LIN {X 0,Y 298.713,Z 404.512,A -85,B 0,C 180,E1 -16393.955,E2 -16393.955} C_VEL
LIN {X 0,Y 299.708,Z 394.679,A -85,B 0,C 180,E1 -16396.344,E2 -16396.344} C_VEL
LIN {X 0,Y 300.926,Z 384.674,A -85,B 0,C 180,E1 -16398.379,E2 -16398.379} C_VEL
LIN {X 0,Y 302.379,Z 372.804,A -85,B 0,C 180,E1 -16400.404,E2 -16400.404} C_VEL
LIN {X 0,Y 303.908,Z 359.25,A -85,B 0,C 180,E1 -16402.329,E2 -16402.329} C_VEL
LIN {X 0,Y 305.452,Z 345.622,A -85,B 0,C 180,E1 -16403.925,E2 -16403.925} C_VEL
LIN {X 0,Y 306.858,Z 331.853,A -85,B 0,C 180,E1 -16405.251,E2 -16405.251} C_VEL
LIN {X 0,Y 308.322,Z 315.885,A -85,B 0,C 180,E1 -16406.482,E2 -16406.482} C_VEL
LIN {X 0,Y 309.428,Z 299.28,A -85,B 0,C 180,E1 -16407.46,E2 -16407.46} C_VEL
LIN {X 0,Y 310.381,Z 282.456,A -85,B 0,C 180,E1 -16408.156,E2 -16408.156} C_VEL
LIN {X 0,Y 315.944,Z 175.453,A -85,B 0,C 180,E1 -16411.633,E2 -16411.633} C_VEL
LIN {X 0,Y 298.499,Z 134.359,A -85,B 0,C 180,E1 -16414.507,E2 -16414.507} C_VEL
LIN {X 0,Y 298.417,Z 133.938,A -85,B 0,C 180,E1 -16414.556,E2 -16414.556} C_VEL
LIN {X 0,Y 298.4,Z 133.941,A -85,B 0,C 180,E1 -16417.761,E2 -16417.761} C_VEL
LIN {X 0,Y 298.349,Z 133.947,A -85,B 0,C 180,E1 -16421.268,E2 -16421.268} C_VEL
LIN {X 0,Y 298.356,Z 133.922,A -85,B 0,C 180,E1 -16425.035,E2 -16425.035} C_VEL
LIN {X 0,Y 298.35,Z 133.935,A -85,B 0,C 180,E1 -16428.921,E2 -16428.921} C_VEL
LIN {X 0,Y 298.4,Z 133.933,A -85,B 0,C 180,E1 -16432.24,E2 -16432.24} C_VEL
LIN {X 0,Y 298.41,Z 133.92,A -85,B 0,C 180,E1 -16435.581,E2 -16435.581} C_VEL
LIN {X 0,Y 298.379,Z 133.936,A -85,B 0,C 180,E1 -16438.789,E2 -16438.789} C_VEL
LIN {X 0,Y 298.413,Z 133.928,A -85,B 0,C 180,E1 -16441.899,E2 -16441.899} C_VEL
LIN {X 0,Y 298.417,Z 133.926,A -85,B 0,C 180,E1 -16444.918,E2 -16444.918} C_VEL
LIN {X 0,Y 298.395,Z 133.941,A -85,B 0,C 180,E1 -16447.862,E2 -16447.862} C_VEL
LIN {X 0,Y 298.463,Z 133.922,A -85,B 0,C 180,E1 -16450.752,E2 -16450.752} C_VEL
LIN {X 0,Y 298.514,Z 133.924,A -85,B 0,C 180,E1 -16454.991,E2 -16454.991} C_VEL
LIN {X 0,Y 298.526,Z 133.999,A -85,B 0,C 180,E1 -16456.297,E2 -16456.297} C_VEL
LIN {X 0,Y 302.475,Z 145.498,A -85,B 0,C 180,E1 -16459.094,E2 -16459.094} C_VEL
LIN {X 0,Y 310.955,Z 161.787,A -85,B 0,C 180,E1 -16460.635,E2 -16460.635} C_VEL
LIN {X 0,Y 320.63,Z 183.073,A -85,B 0,C 180,E1 -16462.347,E2 -16462.347} C_VEL
LIN {X 0,Y 323.385,Z 190.184,A -85,B 0,C 180,E1 -16462.842,E2 -16462.842} C_VEL
LIN {X 0,Y 318.857,Z 312.214,A -85,B 0,C 180,E1 -16465.615,E2 -16465.615} C_VEL
LIN {X 0,Y 317.724,Z 327.891,A -85,B 0,C 180,E1 -16466.195,E2 -16466.195} C_VEL
LIN {X 0,Y 316.387,Z 342.225,A -85,B 0,C 180,E1 -16466.971,E2 -16466.971} C_VEL
LIN {X 0,Y 314.797,Z 355.633,A -85,B 0,C 180,E1 -16467.921,E2 -16467.921} C_VEL
LIN {X 0,Y 312.756,Z 369.748,A -85,B 0,C 180,E1 -16469.195,E2 -16469.195} C_VEL
LIN {X 0,Y 310.496,Z 382.746,A -85,B 0,C 180,E1 -16470.648,E2 -16470.648} C_VEL
LIN {X 0,Y 308.101,Z 395.661,A -85,B 0,C 180,E1 -16472.435,E2 -16472.435} C_VEL
LIN {X 0,Y 305.908,Z 406.678,A -85,B 0,C 180,E1 -16474.282,E2 -16474.282} C_VEL
LIN {X 0,Y 303.719,Z 417.119,A -85,B 0,C 180,E1 -16476.392,E2 -16476.392} C_VEL
LIN {X 0,Y 301.643,Z 426.588,A -85,B 0,C 180,E1 -16478.711,E2 -16478.711} C_VEL
LIN {X 0,Y 300.015,Z 434.716,A -85,B 0,C 180,E1 -16481.143,E2 -16481.143} C_VEL
LIN {X 0,Y 298.703,Z 441.439,A -85,B 0,C 180,E1 -16483.608,E2 -16483.608} C_VEL
LIN {X 0,Y 297.604,Z 447.559,A -85,B 0,C 180,E1 -16486.462,E2 -16486.462} C_VEL
LIN {X 0,Y 297.001,Z 451.472,A -85,B 0,C 180,E1 -16488.82,E2 -16488.82} C_VEL
LIN {X 0,Y 296.584,Z 453.996,A -85,B 0,C 180,E1 -16490.821,E2 -16490.821} C_VEL
LIN {X 0,Y 296.399,Z 455.502,A -85,B 0,C 180,E1 -16492.37,E2 -16492.37} C_VEL
LIN {X 0,Y 296.198,Z 457.301,A -85,B 0,C 180,E1 -16495.283,E2 -16495.283} C_VEL
LIN {X 0,Y 296.215,Z 457.762,A -85,B 0,C 180,E1 -16498.328,E2 -16498.328} C_VEL
LIN {X 0,Y 296.405,Z 456.777,A -85,B 0,C 180,E1 -16501.395,E2 -16501.395} C_VEL
LIN {X 0,Y 296.835,Z 454.759,A -85,B 0,C 180,E1 -16504.036,E2 -16504.036} C_VEL
LIN {X 0,Y 297.466,Z 451.962,A -85,B 0,C 180,E1 -16506.435,E2 -16506.435} C_VEL
LIN {X 0,Y 297.135,Z 450.458,A -85,B 0,C 180,E1 -16507.534,E2 -16507.534} C_VEL
LIN {X 0,Y 294.916,Z 447.714,A -85,B 0,C 180,E1 -16509.328,E2 -16509.328} C_VEL
LIN {X 0,Y 293.14,Z 445.205,A -85,B 0,C 180,E1 -16510.759,E2 -16510.759} C_VEL
LIN {X 0,Y 292.687,Z 443.03,A -85,B 0,C 180,E1 -16511.834,E2 -16511.834} C_VEL
LIN {X 0,Y 292.82,Z 442.243,A -85,B 0,C 180,E1 -16512.189,E2 -16512.189} C_VEL
LIN {X 0,Y 294.596,Z 435.357,A -85,B 0,C 180,E1 -16514.833,E2 -16514.833} C_VEL
LIN {X 0,Y 296.759,Z 427.599,A -85,B 0,C 180,E1 -16517.236,E2 -16517.236} C_VEL
LIN {X 0,Y 298.988,Z 419.592,A -85,B 0,C 180,E1 -16519.294,E2 -16519.294} C_VEL
LIN {X 0,Y 301.649,Z 409.459,A -85,B 0,C 180,E1 -16521.469,E2 -16521.469} C_VEL
LIN {X 0,Y 304.318,Z 398.99,A -85,B 0,C 180,E1 -16523.325,E2 -16523.325} C_VEL
LIN {X 0,Y 307.208,Z 386.777,A -85,B 0,C 180,E1 -16525.115,E2 -16525.115} C_VEL
LIN {X 0,Y 310.013,Z 373.338,A -85,B 0,C 180,E1 -16526.716,E2 -16526.716} C_VEL
LIN {X 0,Y 312.66,Z 358.816,A -85,B 0,C 180,E1 -16528.088,E2 -16528.088} C_VEL
LIN {X 0,Y 314.776,Z 345.041,A -85,B 0,C 180,E1 -16529.101,E2 -16529.101} C_VEL
LIN {X 0,Y 316.458,Z 330.282,A -85,B 0,C 180,E1 -16529.935,E2 -16529.935} C_VEL
LIN {X 0,Y 317.811,Z 314.936,A -85,B 0,C 180,E1 -16530.525,E2 -16530.525} C_VEL
LIN {X 0,Y 318.317,Z 302.146,A -85,B 0,C 180,E1 -16530.882,E2 -16530.882} C_VEL
LIN {X 0,Y 315.448,Z 304.886,A -85,B 0,C 180,E1 -16531.197,E2 -16531.197} C_VEL
LIN {X 0,Y 312.655,Z 306.053,A -85,B 0,C 180,E1 -16531.558,E2 -16531.558} C_VEL
LIN {X 0,Y 311.943,Z 306.129,A -85,B 0,C 180,E1 -16531.659,E2 -16531.659} C_VEL
LIN {X 0,Y 308.747,Z 312.307,A -85,B 0,C 180,E1 -16531.919,E2 -16531.919} C_VEL
LIN {X 0,Y 306.255,Z 315.221,A -85,B 0,C 180,E1 -16532.169,E2 -16532.169} C_VEL
LIN {X 0,Y 304.049,Z 316.166,A -85,B 0,C 180,E1 -16532.464,E2 -16532.464} C_VEL
LIN {X 0,Y 302.853,Z 315.629,A -85,B 0,C 180,E1 -16532.674,E2 -16532.674} C_VEL
LIN {X 0,Y 301.938,Z 313.525,A -85,B 0,C 180,E1 -16532.913,E2 -16532.913} C_VEL
LIN {X 0,Y 301.81,Z 312.672,A -85,B 0,C 180,E1 -16532.994,E2 -16532.994} C_VEL
LIN {X 0,Y 300.389,Z 328.503,A -85,B 0,C 180,E1 -16534.166,E2 -16534.166} C_VEL
LIN {X 0,Y 298.938,Z 342.979,A -85,B 0,C 180,E1 -16535.52,E2 -16535.52} C_VEL
LIN {X 0,Y 297.42,Z 356.501,A -85,B 0,C 180,E1 -16537.065,E2 -16537.065} C_VEL
LIN {X 0,Y 295.874,Z 370.051,A -85,B 0,C 180,E1 -16538.944,E2 -16538.944} C_VEL
LIN {X 0,Y 294.385,Z 381.5,A -85,B 0,C 180,E1 -16540.836,E2 -16540.836} C_VEL
LIN {X 0,Y 293.12,Z 392.122,A -85,B 0,C 180,E1 -16542.919,E2 -16542.919} C_VEL
LIN {X 0,Y 291.957,Z 402.502,A -85,B 0,C 180,E1 -16545.359,E2 -16545.359} C_VEL
LIN {X 0,Y 291.111,Z 410.013,A -85,B 0,C 180,E1 -16547.45,E2 -16547.45} C_VEL
LIN {X 0,Y 290.371,Z 418.242,A -85,B 0,C 180,E1 -16550.245,E2 -16550.245} C_VEL
LIN {X 0,Y 289.956,Z 424.764,A -85,B 0,C 180,E1 -16553.039,E2 -16553.039} C_VEL
LIN {X 0,Y 289.765,Z 429.759,A -85,B 0,C 180,E1 -16555.827,E2 -16555.827} C_VEL
LIN {X 0,Y 289.641,Z 433.363,A -85,B 0,C 180,E1 -16558.609,E2 -16558.609} C_VEL
LIN {X 0,Y 289.791,Z 435.684,A -85,B 0,C 180,E1 -16561.389,E2 -16561.389} C_VEL
LIN {X 0,Y 290.122,Z 436.747,A -85,B 0,C 180,E1 -16564.167,E2 -16564.167} C_VEL
LIN {X 0,Y 290.689,Z 436.577,A -85,B 0,C 180,E1 -16566.943,E2 -16566.943} C_VEL
LIN {X 0,Y 291.75,Z 435.204,A -85,B 0,C 180,E1 -16569.707,E2 -16569.707} C_VEL
LIN {X 0,Y 293.145,Z 432.65,A -85,B 0,C 180,E1 -16572.46,E2 -16572.46} C_VEL
LIN {X 0,Y 294.431,Z 429.964,A -85,B 0,C 180,E1 -16574.515,E2 -16574.515} C_VEL
LIN {X 0,Y 296.723,Z 425.209,A -85,B 0,C 180,E1 -16577.221,E2 -16577.221} C_VEL
LIN {X 0,Y 299.687,Z 419.075,A -85,B 0,C 180,E1 -16579.879,E2 -16579.879} C_VEL
LIN {X 0,Y 303.206,Z 411.451,A -85,B 0,C 180,E1 -16582.485,E2 -16582.485} C_VEL
LIN {X 0,Y 306.675,Z 403.431,A -85,B 0,C 180,E1 -16584.723,E2 -16584.723} C_VEL
LIN {X 0,Y 310.706,Z 393.918,A -85,B 0,C 180,E1 -16586.897,E2 -16586.897} C_VEL
LIN {X 0,Y 315.196,Z 382.723,A -85,B 0,C 180,E1 -16589.003,E2 -16589.003} C_VEL
LIN {X 0,Y 319.857,Z 370.152,A -85,B 0,C 180,E1 -16590.959,E2 -16590.959} C_VEL
LIN {X 0,Y 324.749,Z 355.792,A -85,B 0,C 180,E1 -16592.754,E2 -16592.754} C_VEL
LIN {X 0,Y 328.897,Z 342.374,A -85,B 0,C 180,E1 -16594.119,E2 -16594.119} C_VEL
LIN {X 0,Y 332.878,Z 327.973,A -85,B 0,C 180,E1 -16595.307,E2 -16595.307} C_VEL
LIN {X 0,Y 336.634,Z 312.349,A -85,B 0,C 180,E1 -16596.327,E2 -16596.327} C_VEL
LIN {X 0,Y 339.839,Z 296.318,A -85,B 0,C 180,E1 -16597.128,E2 -16597.128} C_VEL
LIN {X 0,Y 354.117,Z 224.063,A -85,B 0,C 180,E1 -16599.946,E2 -16599.946} C_VEL
LIN {X 0,Y 355.571,Z 217.184,A -85,B 0,C 180,E1 -16600.229,E2 -16600.229} C_VEL
LIN {X 0,Y 354.234,Z 214.83,A -85,B 0,C 180,E1 -16602.1,E2 -16602.1} C_VEL
LIN {X 0,Y 353.367,Z 214.935,A -85,B 0,C 180,E1 -16604.275,E2 -16604.275} C_VEL
LIN {X 0,Y 353.324,Z 216.461,A -85,B 0,C 180,E1 -16605.878,E2 -16605.878} C_VEL
LIN {X 0,Y 353.663,Z 218.476,A -85,B 0,C 180,E1 -16607.134,E2 -16607.134} C_VEL
LIN {X 0,Y 354.272,Z 222.512,A -85,B 0,C 180,E1 -16608.612,E2 -16608.612} C_VEL
LIN {X 0,Y 354.554,Z 224.671,A -85,B 0,C 180,E1 -16609.192,E2 -16609.192} C_VEL
LIN {X 0,Y 340.864,Z 295.02,A -85,B 0,C 180,E1 -16611.907,E2 -16611.907} C_VEL
LIN {X 0,Y 335.929,Z 321.398,A -85,B 0,C 180,E1 -16613,E2 -16613} C_VEL
LIN {X 0,Y 331.767,Z 338.526,A -85,B 0,C 180,E1 -16613.902,E2 -16613.902} C_VEL
LIN {X 0,Y 326.822,Z 355.759,A -85,B 0,C 180,E1 -16615.072,E2 -16615.072} C_VEL
LIN {X 0,Y 321.962,Z 371.081,A -85,B 0,C 180,E1 -16616.41,E2 -16616.41} C_VEL
LIN {X 0,Y 316.965,Z 385.854,A -85,B 0,C 180,E1 -16618.037,E2 -16618.037} C_VEL
LIN {X 0,Y 312.28,Z 398.757,A -85,B 0,C 180,E1 -16619.764,E2 -16619.764} C_VEL
LIN {X 0,Y 307.82,Z 410.76,A -85,B 0,C 180,E1 -16621.722,E2 -16621.722} C_VEL
LIN {X 0,Y 303.56,Z 421.893,A -85,B 0,C 180,E1 -16623.903,E2 -16623.903} C_VEL
LIN {X 0,Y 299.527,Z 432.689,A -85,B 0,C 180,E1 -16626.492,E2 -16626.492} C_VEL
LIN {X 0,Y 296.239,Z 441.705,A -85,B 0,C 180,E1 -16629.154,E2 -16629.154} C_VEL
LIN {X 0,Y 293.617,Z 449.164,A -85,B 0,C 180,E1 -16631.87,E2 -16631.87} C_VEL
LIN {X 0,Y 291.114,Z 459.129,A -85,B 0,C 180,E1 -16636.03,E2 -16636.03} C_VEL
LIN {X 0,Y 290.103,Z 464.483,A -85,B 0,C 180,E1 -16638.825,E2 -16638.825} C_VEL
LIN {X 0,Y 289.628,Z 468.472,A -85,B 0,C 180,E1 -16641.628,E2 -16641.628} C_VEL
LIN {X 0,Y 289.433,Z 471.324,A -85,B 0,C 180,E1 -16644.595,E2 -16644.595} C_VEL
LIN {X 0,Y 289.455,Z 472.691,A -85,B 0,C 180,E1 -16647.217,E2 -16647.217} C_VEL
LIN {X 0,Y 289.439,Z 473.009,A -85,B 0,C 180,E1 -16650,E2 -16650} C_VEL
LIN {X 0,Y 289.481,Z 472.137,A -85,B 0,C 180,E1 -16652.783,E2 -16652.783} C_VEL
LIN {X 0,Y 289.474,Z 470.047,A -85,B 0,C 180,E1 -16655.573,E2 -16655.573} C_VEL
LIN {X 0,Y 289.63,Z 466.684,A -85,B 0,C 180,E1 -16658.372,E2 -16658.372} C_VEL
LIN {X 0,Y 290.017,Z 461.964,A -85,B 0,C 180,E1 -16661.178,E2 -16661.178} C_VEL
LIN {X 0,Y 290.943,Z 456.195,A -85,B 0,C 180,E1 -16663.979,E2 -16663.979} C_VEL
LIN {X 0,Y 292.484,Z 450.761,A -85,B 0,C 180,E1 -16666.759,E2 -16666.759} C_VEL
LIN {X 0,Y 294.74,Z 443.952,A -85,B 0,C 180,E1 -16669.501,E2 -16669.501} C_VEL
LIN {X 0,Y 297.617,Z 435.666,A -85,B 0,C 180,E1 -16672.199,E2 -16672.199} C_VEL
LIN {X 0,Y 301.227,Z 425.689,A -85,B 0,C 180,E1 -16674.832,E2 -16674.832} C_VEL
LIN {X 0,Y 305.188,Z 415.32,A -85,B 0,C 180,E1 -16677.053,E2 -16677.053} C_VEL
LIN {X 0,Y 309.712,Z 403.254,A -85,B 0,C 180,E1 -16679.201,E2 -16679.201} C_VEL
LIN {X 0,Y 314.857,Z 389.006,A -85,B 0,C 180,E1 -16681.263,E2 -16681.263} C_VEL
LIN {X 0,Y 320.273,Z 373.198,A -85,B 0,C 180,E1 -16683.083,E2 -16683.083} C_VEL
LIN {X 0,Y 324.865,Z 358.681,A -85,B 0,C 180,E1 -16684.415,E2 -16684.415} C_VEL
LIN {X 0,Y 329.812,Z 341.583,A -85,B 0,C 180,E1 -16685.639,E2 -16685.639} C_VEL
LIN {X 0,Y 333.873,Z 325.245,A -85,B 0,C 180,E1 -16686.535,E2 -16686.535} C_VEL
LIN {X 0,Y 337.546,Z 307.183,A -85,B 0,C 180,E1 -16687.319,E2 -16687.319} C_VEL
LIN {X 0,Y 350.76,Z 236.513,A -85,B 0,C 180,E1 -16690.093,E2 -16690.093} C_VEL
LIN {X 0,Y 354.605,Z 217.428,A -85,B 0,C 180,E1 -16690.847,E2 -16690.847} C_VEL
LIN {X 0,Y 355.287,Z 213.214,A -85,B 0,C 180,E1 -16691.156,E2 -16691.156} C_VEL
LIN {X 0,Y 354.122,Z 209.776,A -85,B 0,C 180,E1 -16693.001,E2 -16693.001} C_VEL
LIN {X 0,Y 353.446,Z 208.674,A -85,B 0,C 180,E1 -16694.994,E2 -16694.994} C_VEL
LIN {X 0,Y 353.646,Z 208.774,A -85,B 0,C 180,E1 -16696.907,E2 -16696.907} C_VEL
LIN {X 0,Y 354.363,Z 209.968,A -85,B 0,C 180,E1 -16698.38,E2 -16698.38} C_VEL
LIN {X 0,Y 355.341,Z 212.642,A -85,B 0,C 180,E1 -16699.818,E2 -16699.818} C_VEL
LIN {X 0,Y 342.644,Z 276.407,A -85,B 0,C 180,E1 -16702.303,E2 -16702.303} C_VEL
LIN {X 0,Y 338.352,Z 299.721,A -85,B 0,C 180,E1 -16703.24,E2 -16703.24} C_VEL
LIN {X 0,Y 334.973,Z 316.229,A -85,B 0,C 180,E1 -16704.116,E2 -16704.116} C_VEL
LIN {X 0,Y 331.521,Z 330.221,A -85,B 0,C 180,E1 -16705.084,E2 -16705.084} C_VEL
LIN {X 0,Y 327.206,Z 345.754,A -85,B 0,C 180,E1 -16706.422,E2 -16706.422} C_VEL
LIN {X 0,Y 322.441,Z 360.898,A -85,B 0,C 180,E1 -16708.092,E2 -16708.092} C_VEL
LIN {X 0,Y 317.943,Z 373.671,A -85,B 0,C 180,E1 -16709.809,E2 -16709.809} C_VEL
LIN {X 0,Y 313.195,Z 386.308,A -85,B 0,C 180,E1 -16711.886,E2 -16711.886} C_VEL
LIN {X 0,Y 308.878,Z 396.966,A -85,B 0,C 180,E1 -16714.024,E2 -16714.024} C_VEL
LIN {X 0,Y 305.074,Z 405.94,A -85,B 0,C 180,E1 -16716.225,E2 -16716.225} C_VEL
LIN {X 0,Y 301.728,Z 413.725,A -85,B 0,C 180,E1 -16718.571,E2 -16718.571} C_VEL
LIN {X 0,Y 298.865,Z 419.817,A -85,B 0,C 180,E1 -16720.779,E2 -16720.779} C_VEL
LIN {X 0,Y 296.031,Z 425.703,A -85,B 0,C 180,E1 -16723.448,E2 -16723.448} C_VEL
LIN {X 0,Y 293.902,Z 430.203,A -85,B 0,C 180,E1 -16726.165,E2 -16726.165} C_VEL
LIN {X 0,Y 292.409,Z 433.42,A -85,B 0,C 180,E1 -16728.915,E2 -16728.915} C_VEL
LIN {X 0,Y 290.94,Z 435.639,A -85,B 0,C 180,E1 -16732.056,E2 -16732.056} C_VEL
LIN {X 0,Y 290.278,Z 436.299,A -85,B 0,C 180,E1 -16734.443,E2 -16734.443} C_VEL
LIN {X 0,Y 289.943,Z 435.9,A -85,B 0,C 180,E1 -16737.222,E2 -16737.222} C_VEL
LIN {X 0,Y 289.666,Z 434.263,A -85,B 0,C 180,E1 -16740,E2 -16740} C_VEL
LIN {X 0,Y 289.67,Z 431.361,A -85,B 0,C 180,E1 -16742.782,E2 -16742.782} C_VEL
LIN {X 0,Y 289.788,Z 427.115,A -85,B 0,C 180,E1 -16745.567,E2 -16745.567} C_VEL
LIN {X 0,Y 290.137,Z 421.423,A -85,B 0,C 180,E1 -16748.357,E2 -16748.357} C_VEL
LIN {X 0,Y 290.663,Z 414.127,A -85,B 0,C 180,E1 -16751.154,E2 -16751.154} C_VEL
LIN {X 0,Y 291.53,Z 406.214,A -85,B 0,C 180,E1 -16753.595,E2 -16753.595} C_VEL
LIN {X 0,Y 292.345,Z 397.131,A -85,B 0,C 180,E1 -16755.929,E2 -16755.929} C_VEL
LIN {X 0,Y 293.605,Z 386.89,A -85,B 0,C 180,E1 -16758.131,E2 -16758.131} C_VEL
LIN {X 0,Y 295.175,Z 374.325,A -85,B 0,C 180,E1 -16760.379,E2 -16760.379} C_VEL
LIN {X 0,Y 296.656,Z 361.542,A -85,B 0,C 180,E1 -16762.275,E2 -16762.275} C_VEL
LIN {X 0,Y 298.335,Z 347.669,A -85,B 0,C 180,E1 -16763.977,E2 -16763.977} C_VEL
LIN {X 0,Y 299.907,Z 332.376,A -85,B 0,C 180,E1 -16765.506,E2 -16765.506} C_VEL
LIN {X 0,Y 301.397,Z 316.461,A -85,B 0,C 180,E1 -16766.765,E2 -16766.765} C_VEL
LIN {X 0,Y 302.554,Z 300.04,A -85,B 0,C 180,E1 -16767.762,E2 -16767.762} C_VEL
LIN {X 0,Y 303.532,Z 282.966,A -85,B 0,C 180,E1 -16768.493,E2 -16768.493} C_VEL
LIN {X 0,Y 309.088,Z 176.89,A -85,B 0,C 180,E1 -16772.068,E2 -16772.068} C_VEL
LIN {X 0,Y 291.493,Z 135.429,A -85,B 0,C 180,E1 -16775.049,E2 -16775.049} C_VEL
LIN {X 0,Y 291.386,Z 134.814,A -85,B 0,C 180,E1 -16775.128,E2 -16775.128} C_VEL
LIN {X 0,Y 291.336,Z 134.82,A -85,B 0,C 180,E1 -16778.845,E2 -16778.845} C_VEL
LIN {X 0,Y 291.289,Z 134.825,A -85,B 0,C 180,E1 -16782.499,E2 -16782.499} C_VEL
LIN {X 0,Y 291.29,Z 134.79,A -85,B 0,C 180,E1 -16786.371,E2 -16786.371} C_VEL
LIN {X 0,Y 291.358,Z 134.817,A -85,B 0,C 180,E1 -16790.525,E2 -16790.525} C_VEL
LIN {X 0,Y 291.392,Z 134.794,A -85,B 0,C 180,E1 -16792.917,E2 -16792.917} C_VEL
LIN {X 0,Y 291.346,Z 134.812,A -85,B 0,C 180,E1 -16796.302,E2 -16796.302} C_VEL
LIN {X 0,Y 291.367,Z 134.796,A -85,B 0,C 180,E1 -16800.268,E2 -16800.268} C_VEL
LIN {X 0,Y 291.346,Z 134.815,A -85,B 0,C 180,E1 -16804.265,E2 -16804.265} C_VEL
LIN {X 0,Y 291.353,Z 134.812,A -85,B 0,C 180,E1 -16807.297,E2 -16807.297} C_VEL
LIN {X 0,Y 291.388,Z 134.801,A -85,B 0,C 180,E1 -16810.265,E2 -16810.265} C_VEL
LIN {X 0,Y 291.477,Z 134.797,A -85,B 0,C 180,E1 -16814.683,E2 -16814.683} C_VEL
LIN {X 0,Y 291.515,Z 135.005,A -85,B 0,C 180,E1 -16815.461,E2 -16815.461} C_VEL
LIN {X 0,Y 295.251,Z 145.74,A -85,B 0,C 180,E1 -16818.133,E2 -16818.133} C_VEL
LIN {X 0,Y 303.967,Z 162.064,A -85,B 0,C 180,E1 -16819.777,E2 -16819.777} C_VEL
LIN {X 0,Y 311.708,Z 178.744,A -85,B 0,C 180,E1 -16821.207,E2 -16821.207} C_VEL
LIN {X 0,Y 316.237,Z 189.177,A -85,B 0,C 180,E1 -16822.02,E2 -16822.02} C_VEL
LIN {X 0,Y 317.229,Z 191.723,A -85,B 0,C 180,E1 -16822.201,E2 -16822.201} C_VEL
LIN {X 0,Y 312.632,Z 312.524,A -85,B 0,C 180,E1 -16825.003,E2 -16825.003} C_VEL
LIN {X 0,Y 311.48,Z 328.136,A -85,B 0,C 180,E1 -16825.592,E2 -16825.592} C_VEL
LIN {X 0,Y 310.038,Z 342.988,A -85,B 0,C 180,E1 -16826.416,E2 -16826.416} C_VEL
LIN {X 0,Y 308.365,Z 356.344,A -85,B 0,C 180,E1 -16827.387,E2 -16827.387} C_VEL
LIN {X 0,Y 306.486,Z 368.83,A -85,B 0,C 180,E1 -16828.522,E2 -16828.522} C_VEL
LIN {X 0,Y 304.158,Z 382.017,A -85,B 0,C 180,E1 -16830,E2 -16830} C_VEL
LIN {X 0,Y 301.851,Z 394.123,A -85,B 0,C 180,E1 -16831.668,E2 -16831.668} C_VEL
LIN {X 0,Y 299.363,Z 406.237,A -85,B 0,C 180,E1 -16833.702,E2 -16833.702} C_VEL
LIN {X 0,Y 297.026,Z 416.893,A -85,B 0,C 180,E1 -16835.879,E2 -16835.879} C_VEL
LIN {X 0,Y 294.912,Z 426.333,A -85,B 0,C 180,E1 -16838.221,E2 -16838.221} C_VEL
LIN {X 0,Y 293.219,Z 434.431,A -85,B 0,C 180,E1 -16840.668,E2 -16840.668} C_VEL
LIN {X 0,Y 291.777,Z 441.338,A -85,B 0,C 180,E1 -16843.228,E2 -16843.228} C_VEL
LIN {X 0,Y 290.63,Z 447.519,A -85,B 0,C 180,E1 -16846.146,E2 -16846.146} C_VEL
LIN {X 0,Y 289.864,Z 452.068,A -85,B 0,C 180,E1 -16848.986,E2 -16848.986} C_VEL
LIN {X 0,Y 289.426,Z 454.825,A -85,B 0,C 180,E1 -16851.361,E2 -16851.361} C_VEL
LIN {X 0,Y 289.118,Z 457.097,A -85,B 0,C 180,E1 -16854.409,E2 -16854.409} C_VEL
LIN {X 0,Y 289.062,Z 457.98,A -85,B 0,C 180,E1 -16857.513,E2 -16857.513} C_VEL
LIN {X 0,Y 289.14,Z 457.886,A -85,B 0,C 180,E1 -16859.087,E2 -16859.087} C_VEL
LIN {X 0,Y 289.338,Z 456.855,A -85,B 0,C 180,E1 -16861.771,E2 -16861.771} C_VEL
LIN {X 0,Y 289.815,Z 454.76,A -85,B 0,C 180,E1 -16864.461,E2 -16864.461} C_VEL
LIN {X 0,Y 290.583,Z 451.479,A -85,B 0,C 180,E1 -16867.203,E2 -16867.203} C_VEL
LIN {X 0,Y 291.485,Z 447.781,A -85,B 0,C 180,E1 -16869.506,E2 -16869.506} C_VEL
LIN {X 0,Y 292.82,Z 442.243,A -85,B 0,C 180,E1 -16872.189,E2 -16872.189} C_VEL
LIN {X 0,Y 292.83,Z 439.86,A -85,B 0,C 180,E1 -16873.248,E2 -16873.248} C_VEL
LIN {X 0,Y 291.178,Z 435.782,A -85,B 0,C 180,E1 -16874.994,E2 -16874.994} C_VEL
LIN {X 0,Y 289.746,Z 431.245,A -85,B 0,C 180,E1 -16876.71,E2 -16876.71} C_VEL
LIN {X 0,Y 290.086,Z 428.105,A -85,B 0,C 180,E1 -16877.697,E2 -16877.697} C_VEL
LIN {X 0,Y 292.862,Z 418.618,A -85,B 0,C 180,E1 -16880.168,E2 -16880.168} C_VEL
LIN {X 0,Y 295.781,Z 407.846,A -85,B 0,C 180,E1 -16882.469,E2 -16882.469} C_VEL
LIN {X 0,Y 298.778,Z 396.667,A -85,B 0,C 180,E1 -16884.407,E2 -16884.407} C_VEL
LIN {X 0,Y 301.634,Z 384.763,A -85,B 0,C 180,E1 -16886.113,E2 -16886.113} C_VEL
LIN {X 0,Y 304.177,Z 373.032,A -85,B 0,C 180,E1 -16887.494,E2 -16887.494} C_VEL
LIN {X 0,Y 306.874,Z 358.626,A -85,B 0,C 180,E1 -16888.866,E2 -16888.866} C_VEL
LIN {X 0,Y 309.158,Z 343.968,A -85,B 0,C 180,E1 -16889.945,E2 -16889.945} C_VEL
LIN {X 0,Y 310.965,Z 328.633,A -85,B 0,C 180,E1 -16890.79,E2 -16890.79} C_VEL
LIN {X 0,Y 311.922,Z 318.051,A -85,B 0,C 180,E1 -16891.209,E2 -16891.209} C_VEL
LIN {X 0,Y 311.3,Z 318.381,A -85,B 0,C 180,E1 -16891.285,E2 -16891.285} C_VEL
LIN {X 0,Y 307.831,Z 321.576,A -85,B 0,C 180,E1 -16891.638,E2 -16891.638} C_VEL
LIN {X 0,Y 304.902,Z 322.888,A -85,B 0,C 180,E1 -16892.006,E2 -16892.006} C_VEL
LIN {X 0,Y 302.532,Z 323.456,A -85,B 0,C 180,E1 -16892.338,E2 -16892.338} C_VEL
LIN {X 0,Y 299.211,Z 327.365,A -85,B 0,C 180,E1 -16892.637,E2 -16892.637} C_VEL
LIN {X 0,Y 297.173,Z 328.653,A -85,B 0,C 180,E1 -16892.88,E2 -16892.88} C_VEL
LIN {X 0,Y 295.205,Z 328.719,A -85,B 0,C 180,E1 -16893.201,E2 -16893.201} C_VEL
LIN {X 0,Y 294.197,Z 327.728,A -85,B 0,C 180,E1 -16893.437,E2 -16893.437} C_VEL
LIN {X 0,Y 293.728,Z 325.806,A -85,B 0,C 180,E1 -16893.631,E2 -16893.631} C_VEL
LIN {X 0,Y 292.16,Z 341.721,A -85,B 0,C 180,E1 -16895.104,E2 -16895.104} C_VEL
LIN {X 0,Y 290.63,Z 355.402,A -85,B 0,C 180,E1 -16896.668,E2 -16896.668} C_VEL
LIN {X 0,Y 288.967,Z 369.319,A -85,B 0,C 180,E1 -16898.603,E2 -16898.603} C_VEL
LIN {X 0,Y 287.315,Z 381.897,A -85,B 0,C 180,E1 -16900.717,E2 -16900.717} C_VEL
LIN {X 0,Y 286.041,Z 392.523,A -85,B 0,C 180,E1 -16902.852,E2 -16902.852} C_VEL
LIN {X 0,Y 285.011,Z 401.571,A -85,B 0,C 180,E1 -16904.994,E2 -16904.994} C_VEL
LIN {X 0,Y 284.001,Z 410.42,A -85,B 0,C 180,E1 -16907.494,E2 -16907.494} C_VEL
LIN {X 0,Y 283.34,Z 417.756,A -85,B 0,C 180,E1 -16910.001,E2 -16910.001} C_VEL
LIN {X 0,Y 282.892,Z 424.499,A -85,B 0,C 180,E1 -16912.864,E2 -16912.864} C_VEL
LIN {X 0,Y 282.678,Z 429.684,A -85,B 0,C 180,E1 -16915.722,E2 -16915.722} C_VEL
LIN {X 0,Y 282.556,Z 433.461,A -85,B 0,C 180,E1 -16918.574,E2 -16918.574} C_VEL
LIN {X 0,Y 282.702,Z 435.923,A -85,B 0,C 180,E1 -16921.424,E2 -16921.424} C_VEL
LIN {X 0,Y 283.053,Z 437.152,A -85,B 0,C 180,E1 -16924.271,E2 -16924.271} C_VEL
LIN {X 0,Y 283.686,Z 437.178,A -85,B 0,C 180,E1 -16927.115,E2 -16927.115} C_VEL
LIN {X 0,Y 284.784,Z 436.017,A -85,B 0,C 180,E1 -16929.947,E2 -16929.947} C_VEL
LIN {X 0,Y 286.279,Z 433.682,A -85,B 0,C 180,E1 -16932.764,E2 -16932.764} C_VEL
LIN {X 0,Y 288.264,Z 430.14,A -85,B 0,C 180,E1 -16935.556,E2 -16935.556} C_VEL
LIN {X 0,Y 290.796,Z 425.319,A -85,B 0,C 180,E1 -16938.311,E2 -16938.311} C_VEL
LIN {X 0,Y 294.155,Z 419.088,A -85,B 0,C 180,E1 -16941.001,E2 -16941.001} C_VEL
LIN {X 0,Y 297.923,Z 411.43,A -85,B 0,C 180,E1 -16943.642,E2 -16943.642} C_VEL
LIN {X 0,Y 301.752,Z 403.352,A -85,B 0,C 180,E1 -16945.893,E2 -16945.893} C_VEL
LIN {X 0,Y 306.117,Z 393.831,A -85,B 0,C 180,E1 -16948.076,E2 -16948.076} C_VEL
LIN {X 0,Y 310.934,Z 382.639,A -85,B 0,C 180,E1 -16950.193,E2 -16950.193} C_VEL
LIN {X 0,Y 315.713,Z 370.709,A -85,B 0,C 180,E1 -16952.048,E2 -16952.048} C_VEL
LIN {X 0,Y 321.191,Z 355.801,A -85,B 0,C 180,E1 -16953.915,E2 -16953.915} C_VEL
LIN {X 0,Y 326.011,Z 341.146,A -85,B 0,C 180,E1 -16955.405,E2 -16955.405} C_VEL
LIN {X 0,Y 330.827,Z 324.799,A -85,B 0,C 180,E1 -16956.689,E2 -16956.689} C_VEL
LIN {X 0,Y 334.812,Z 308.55,A -85,B 0,C 180,E1 -16957.688,E2 -16957.688} C_VEL
LIN {X 0,Y 337.923,Z 293.646,A -85,B 0,C 180,E1 -16958.365,E2 -16958.365} C_VEL
LIN {X 0,Y 352.283,Z 225.795,A -85,B 0,C 180,E1 -16961.022,E2 -16961.022} C_VEL
LIN {X 0,Y 352.912,Z 222.988,A -85,B 0,C 180,E1 -16961.132,E2 -16961.132} C_VEL
LIN {X 0,Y 352.217,Z 221.574,A -85,B 0,C 180,E1 -16962.415,E2 -16962.415} C_VEL
LIN {X 0,Y 351.517,Z 221.916,A -85,B 0,C 180,E1 -16964.408,E2 -16964.408} C_VEL
LIN {X 0,Y 351.495,Z 223.639,A -85,B 0,C 180,E1 -16966.038,E2 -16966.038} C_VEL
LIN {X 0,Y 351.683,Z 225.422,A -85,B 0,C 180,E1 -16966.984,E2 -16966.984} C_VEL
LIN {X 0,Y 352.054,Z 228.809,A -85,B 0,C 180,E1 -16968.213,E2 -16968.213} C_VEL
LIN {X 0,Y 338.078,Z 296.297,A -85,B 0,C 180,E1 -16970.822,E2 -16970.822} C_VEL
LIN {X 0,Y 332.994,Z 321.336,A -85,B 0,C 180,E1 -16971.878,E2 -16971.878} C_VEL
LIN {X 0,Y 328.425,Z 338.716,A -85,B 0,C 180,E1 -16972.805,E2 -16972.805} C_VEL
LIN {X 0,Y 323.504,Z 354.737,A -85,B 0,C 180,E1 -16973.894,E2 -16973.894} C_VEL
LIN {X 0,Y 318.456,Z 369.573,A -85,B 0,C 180,E1 -16975.178,E2 -16975.178} C_VEL
LIN {X 0,Y 313.435,Z 383.381,A -85,B 0,C 180,E1 -16976.677,E2 -16976.677} C_VEL
LIN {X 0,Y 307.987,Z 397.41,A -85,B 0,C 180,E1 -16978.534,E2 -16978.534} C_VEL
LIN {X 0,Y 303.141,Z 409.406,A -85,B 0,C 180,E1 -16980.484,E2 -16980.484} C_VEL
LIN {X 0,Y 297.952,Z 422.007,A -85,B 0,C 180,E1 -16982.995,E2 -16982.995} C_VEL
LIN {X 0,Y 293.528,Z 432.761,A -85,B 0,C 180,E1 -16985.664,E2 -16985.664} C_VEL
LIN {X 0,Y 290.026,Z 441.457,A -85,B 0,C 180,E1 -16988.313,E2 -16988.313} C_VEL
LIN {X 0,Y 286.881,Z 449.616,A -85,B 0,C 180,E1 -16991.429,E2 -16991.429} C_VEL
LIN {X 0,Y 283.889,Z 460.526,A -85,B 0,C 180,E1 -16996.398,E2 -16996.398} C_VEL
LIN {X 0,Y 282.938,Z 465.478,A -85,B 0,C 180,E1 -16999.263,E2 -16999.263} C_VEL
LIN {X 0,Y 282.564,Z 468.362,A -85,B 0,C 180,E1 -17001.417,E2 -17001.417} C_VEL
LIN {X 0,Y 282.376,Z 471.049,A -85,B 0,C 180,E1 -17004.286,E2 -17004.286} C_VEL
LIN {X 0,Y 282.359,Z 472.527,A -85,B 0,C 180,E1 -17007.147,E2 -17007.147} C_VEL
LIN {X 0,Y 282.359,Z 472.816,A -85,B 0,C 180,E1 -17010,E2 -17010} C_VEL
LIN {X 0,Y 282.383,Z 471.913,A -85,B 0,C 180,E1 -17012.853,E2 -17012.853} C_VEL
LIN {X 0,Y 282.381,Z 469.79,A -85,B 0,C 180,E1 -17015.713,E2 -17015.713} C_VEL
LIN {X 0,Y 282.567,Z 466.393,A -85,B 0,C 180,E1 -17018.582,E2 -17018.582} C_VEL
LIN {X 0,Y 282.989,Z 461.638,A -85,B 0,C 180,E1 -17021.46,E2 -17021.46} C_VEL
LIN {X 0,Y 283.713,Z 457.422,A -85,B 0,C 180,E1 -17023.611,E2 -17023.611} C_VEL
LIN {X 0,Y 285.177,Z 452.563,A -85,B 0,C 180,E1 -17026.464,E2 -17026.464} C_VEL
LIN {X 0,Y 287.411,Z 446.359,A -85,B 0,C 180,E1 -17029.276,E2 -17029.276} C_VEL
LIN {X 0,Y 290.311,Z 438.728,A -85,B 0,C 180,E1 -17032.039,E2 -17032.039} C_VEL
LIN {X 0,Y 293.401,Z 430.966,A -85,B 0,C 180,E1 -17034.37,E2 -17034.37} C_VEL
LIN {X 0,Y 297.225,Z 421.589,A -85,B 0,C 180,E1 -17036.696,E2 -17036.696} C_VEL
LIN {X 0,Y 301.696,Z 410.738,A -85,B 0,C 180,E1 -17038.906,E2 -17038.906} C_VEL
LIN {X 0,Y 306.754,Z 398.122,A -85,B 0,C 180,E1 -17041.031,E2 -17041.031} C_VEL
LIN {X 0,Y 312.117,Z 384.303,A -85,B 0,C 180,E1 -17042.904,E2 -17042.904} C_VEL
LIN {X 0,Y 317.486,Z 369.305,A -85,B 0,C 180,E1 -17044.558,E2 -17044.558} C_VEL
LIN {X 0,Y 322.522,Z 354.378,A -85,B 0,C 180,E1 -17045.847,E2 -17045.847} C_VEL
LIN {X 0,Y 327.394,Z 338.338,A -85,B 0,C 180,E1 -17046.946,E2 -17046.946} C_VEL
LIN {X 0,Y 331.683,Z 321.692,A -85,B 0,C 180,E1 -17047.818,E2 -17047.818} C_VEL
LIN {X 0,Y 336.282,Z 299.102,A -85,B 0,C 180,E1 -17048.779,E2 -17048.779} C_VEL
LIN {X 0,Y 351.164,Z 226.425,A -85,B 0,C 180,E1 -17051.615,E2 -17051.615} C_VEL
LIN {X 0,Y 352.747,Z 218.942,A -85,B 0,C 180,E1 -17051.938,E2 -17051.938} C_VEL
LIN {X 0,Y 352.716,Z 218.449,A -85,B 0,C 180,E1 -17052.08,E2 -17052.08} C_VEL
LIN {X 0,Y 352.126,Z 216.458,A -85,B 0,C 180,E1 -17053.305,E2 -17053.305} C_VEL
LIN {X 0,Y 351.652,Z 215.533,A -85,B 0,C 180,E1 -17055.003,E2 -17055.003} C_VEL
LIN {X 0,Y 351.846,Z 215.654,A -85,B 0,C 180,E1 -17056.91,E2 -17056.91} C_VEL
LIN {X 0,Y 352.419,Z 216.827,A -85,B 0,C 180,E1 -17058.239,E2 -17058.239} C_VEL
LIN {X 0,Y 352.774,Z 217.97,A -85,B 0,C 180,E1 -17058.896,E2 -17058.896} C_VEL
LIN {X 0,Y 337.935,Z 288.589,A -85,B 0,C 180,E1 -17061.636,E2 -17061.636} C_VEL
LIN {X 0,Y 334.291,Z 306.792,A -85,B 0,C 180,E1 -17062.434,E2 -17062.434} C_VEL
LIN {X 0,Y 330.817,Z 321.513,A -85,B 0,C 180,E1 -17063.309,E2 -17063.309} C_VEL
LIN {X 0,Y 326.512,Z 336.946,A -85,B 0,C 180,E1 -17064.468,E2 -17064.468} C_VEL
LIN {X 0,Y 321.99,Z 351.095,A -85,B 0,C 180,E1 -17065.803,E2 -17065.803} C_VEL
LIN {X 0,Y 317.059,Z 365.361,A -85,B 0,C 180,E1 -17067.484,E2 -17067.484} C_VEL
LIN {X 0,Y 311.875,Z 378.778,A -85,B 0,C 180,E1 -17069.439,E2 -17069.439} C_VEL
LIN {X 0,Y 306.729,Z 390.928,A -85,B 0,C 180,E1 -17071.612,E2 -17071.612} C_VEL
LIN {X 0,Y 302.293,Z 400.844,A -85,B 0,C 180,E1 -17073.786,E2 -17073.786} C_VEL
LIN {X 0,Y 298.374,Z 409.229,A -85,B 0,C 180,E1 -17076.027,E2 -17076.027} C_VEL
LIN {X 0,Y 294.776,Z 416.752,A -85,B 0,C 180,E1 -17078.501,E2 -17078.501} C_VEL
LIN {X 0,Y 291.571,Z 422.965,A -85,B 0,C 180,E1 -17081.01,E2 -17081.01} C_VEL
LIN {X 0,Y 288.765,Z 428.238,A -85,B 0,C 180,E1 -17083.747,E2 -17083.747} C_VEL
LIN {X 0,Y 287.096,Z 431.327,A -85,B 0,C 180,E1 -17085.831,E2 -17085.831} C_VEL
LIN {X 0,Y 285.495,Z 434.319,A -85,B 0,C 180,E1 -17088.643,E2 -17088.643} C_VEL
LIN {X 0,Y 283.904,Z 436.372,A -85,B 0,C 180,E1 -17091.97,E2 -17091.97} C_VEL
LIN {X 0,Y 283.243,Z 436.789,A -85,B 0,C 180,E1 -17094.304,E2 -17094.304} C_VEL
LIN {X 0,Y 282.859,Z 436.215,A -85,B 0,C 180,E1 -17097.152,E2 -17097.152} C_VEL
LIN {X 0,Y 282.576,Z 434.427,A -85,B 0,C 180,E1 -17100,E2 -17100} C_VEL
LIN {X 0,Y 282.593,Z 431.363,A -85,B 0,C 180,E1 -17102.851,E2 -17102.851} C_VEL
LIN {X 0,Y 282.7,Z 426.93,A -85,B 0,C 180,E1 -17105.707,E2 -17105.707} C_VEL
LIN {X 0,Y 282.952,Z 422.617,A -85,B 0,C 180,E1 -17107.852,E2 -17107.852} C_VEL
LIN {X 0,Y 283.45,Z 415.502,A -85,B 0,C 180,E1 -17110.718,E2 -17110.718} C_VEL
LIN {X 0,Y 284.265,Z 407.795,A -85,B 0,C 180,E1 -17113.221,E2 -17113.221} C_VEL
LIN {X 0,Y 285,Z 399.902,A -85,B 0,C 180,E1 -17115.373,E2 -17115.373} C_VEL
LIN {X 0,Y 286.294,Z 388.963,A -85,B 0,C 180,E1 -17117.87,E2 -17117.87} C_VEL
LIN {X 0,Y 287.703,Z 377.767,A -85,B 0,C 180,E1 -17119.999,E2 -17119.999} C_VEL
LIN {X 0,Y 289.232,Z 365.597,A -85,B 0,C 180,E1 -17121.938,E2 -17121.938} C_VEL
LIN {X 0,Y 290.981,Z 351.324,A -85,B 0,C 180,E1 -17123.826,E2 -17123.826} C_VEL
LIN {X 0,Y 292.584,Z 336.458,A -85,B 0,C 180,E1 -17125.428,E2 -17125.428} C_VEL
LIN {X 0,Y 294.195,Z 320.336,A -85,B 0,C 180,E1 -17126.802,E2 -17126.802} C_VEL
LIN {X 0,Y 295.422,Z 304.075,A -85,B 0,C 180,E1 -17127.88,E2 -17127.88} C_VEL
LIN {X 0,Y 296.429,Z 287.373,A -85,B 0,C 180,E1 -17128.69,E2 -17128.69} C_VEL
LIN {X 0,Y 302.438,Z 178.79,A -85,B 0,C 180,E1 -17132.469,E2 -17132.469} C_VEL
LIN {X 0,Y 284.469,Z 136.374,A -85,B 0,C 180,E1 -17135.604,E2 -17135.604} C_VEL
LIN {X 0,Y 284.343,Z 135.692,A -85,B 0,C 180,E1 -17135.683,E2 -17135.683} C_VEL
LIN {X 0,Y 284.283,Z 135.699,A -85,B 0,C 180,E1 -17139.999,E2 -17139.999} C_VEL
LIN {X 0,Y 284.236,Z 135.695,A -85,B 0,C 180,E1 -17144.188,E2 -17144.188} C_VEL
LIN {X 0,Y 284.241,Z 135.678,A -85,B 0,C 180,E1 -17148.119,E2 -17148.119} C_VEL
LIN {X 0,Y 284.31,Z 135.686,A -85,B 0,C 180,E1 -17152.282,E2 -17152.282} C_VEL
LIN {X 0,Y 284.309,Z 135.672,A -85,B 0,C 180,E1 -17155.351,E2 -17155.351} C_VEL
LIN {X 0,Y 284.287,Z 135.692,A -85,B 0,C 180,E1 -17158.725,E2 -17158.725} C_VEL
LIN {X 0,Y 284.284,Z 135.688,A -85,B 0,C 180,E1 -17161.984,E2 -17161.984} C_VEL
LIN {X 0,Y 284.295,Z 135.68,A -85,B 0,C 180,E1 -17166.16,E2 -17166.16} C_VEL
LIN {X 0,Y 284.336,Z 135.679,A -85,B 0,C 180,E1 -17169.928,E2 -17169.928} C_VEL
LIN {X 0,Y 284.433,Z 135.735,A -85,B 0,C 180,E1 -17174.505,E2 -17174.505} C_VEL
LIN {X 0,Y 288.047,Z 145.899,A -85,B 0,C 180,E1 -17177.118,E2 -17177.118} C_VEL
LIN {X 0,Y 298.355,Z 165.025,A -85,B 0,C 180,E1 -17179.138,E2 -17179.138} C_VEL
LIN {X 0,Y 306.153,Z 181.921,A -85,B 0,C 180,E1 -17180.63,E2 -17180.63} C_VEL
LIN {X 0,Y 311.117,Z 193.551,A -85,B 0,C 180,E1 -17181.556,E2 -17181.556} C_VEL
LIN {X 0,Y 306.439,Z 312.604,A -85,B 0,C 180,E1 -17184.365,E2 -17184.365} C_VEL
LIN {X 0,Y 305.234,Z 328.28,A -85,B 0,C 180,E1 -17184.964,E2 -17184.964} C_VEL
LIN {X 0,Y 303.826,Z 342.664,A -85,B 0,C 180,E1 -17185.772,E2 -17185.772} C_VEL
LIN {X 0,Y 301.884,Z 357.335,A -85,B 0,C 180,E1 -17186.859,E2 -17186.859} C_VEL
LIN {X 0,Y 299.794,Z 370.922,A -85,B 0,C 180,E1 -17188.153,E2 -17188.153} C_VEL
LIN {X 0,Y 297.37,Z 383.807,A -85,B 0,C 180,E1 -17189.661,E2 -17189.661} C_VEL
LIN {X 0,Y 294.975,Z 395.688,A -85,B 0,C 180,E1 -17191.365,E2 -17191.365} C_VEL
LIN {X 0,Y 292.441,Z 407.569,A -85,B 0,C 180,E1 -17193.444,E2 -17193.444} C_VEL
LIN {X 0,Y 290.152,Z 417.58,A -85,B 0,C 180,E1 -17195.56,E2 -17195.56} C_VEL
LIN {X 0,Y 287.886,Z 427.331,A -85,B 0,C 180,E1 -17198.069,E2 -17198.069} C_VEL
LIN {X 0,Y 286.076,Z 435.573,A -85,B 0,C 180,E1 -17200.678,E2 -17200.678} C_VEL
LIN {X 0,Y 284.518,Z 442.896,A -85,B 0,C 180,E1 -17203.572,E2 -17203.572} C_VEL
LIN {X 0,Y 283.39,Z 448.778,A -85,B 0,C 180,E1 -17206.571,E2 -17206.571} C_VEL
LIN {X 0,Y 282.719,Z 452.626,A -85,B 0,C 180,E1 -17209.155,E2 -17209.155} C_VEL
LIN {X 0,Y 282.27,Z 455.606,A -85,B 0,C 180,E1 -17211.93,E2 -17211.93} C_VEL
LIN {X 0,Y 282,Z 457.585,A -85,B 0,C 180,E1 -17215.067,E2 -17215.067} C_VEL
LIN {X 0,Y 281.997,Z 458.163,A -85,B 0,C 180,E1 -17218.263,E2 -17218.263} C_VEL
LIN {X 0,Y 282.077,Z 457.906,A -85,B 0,C 180,E1 -17219.888,E2 -17219.888} C_VEL
LIN {X 0,Y 282.305,Z 456.93,A -85,B 0,C 180,E1 -17222.173,E2 -17222.173} C_VEL
LIN {X 0,Y 282.846,Z 454.754,A -85,B 0,C 180,E1 -17224.918,E2 -17224.918} C_VEL
LIN {X 0,Y 283.589,Z 451.674,A -85,B 0,C 180,E1 -17227.529,E2 -17227.529} C_VEL
LIN {X 0,Y 284.634,Z 447.694,A -85,B 0,C 180,E1 -17230.054,E2 -17230.054} C_VEL
LIN {X 0,Y 286.168,Z 441.909,A -85,B 0,C 180,E1 -17232.872,E2 -17232.872} C_VEL
LIN {X 0,Y 288.065,Z 435.008,A -85,B 0,C 180,E1 -17235.53,E2 -17235.53} C_VEL
LIN {X 0,Y 290.086,Z 428.105,A -85,B 0,C 180,E1 -17237.697,E2 -17237.697} C_VEL
LIN {X 0,Y 290.492,Z 424.858,A -85,B 0,C 180,E1 -17238.669,E2 -17238.669} C_VEL
LIN {X 0,Y 289.455,Z 419.522,A -85,B 0,C 180,E1 -17240.31,E2 -17240.31} C_VEL
LIN {X 0,Y 288.495,Z 413.78,A -85,B 0,C 180,E1 -17241.902,E2 -17241.902} C_VEL
LIN {X 0,Y 289.001,Z 409.88,A -85,B 0,C 180,E1 -17242.778,E2 -17242.778} C_VEL
LIN {X 0,Y 292.217,Z 398.453,A -85,B 0,C 180,E1 -17244.857,E2 -17244.857} C_VEL
LIN {X 0,Y 295.348,Z 386.047,A -85,B 0,C 180,E1 -17246.705,E2 -17246.705} C_VEL
LIN {X 0,Y 298.274,Z 373.185,A -85,B 0,C 180,E1 -17248.258,E2 -17248.258} C_VEL
LIN {X 0,Y 300.925,Z 359.677,A -85,B 0,C 180,E1 -17249.573,E2 -17249.573} C_VEL
LIN {X 0,Y 303.199,Z 346.115,A -85,B 0,C 180,E1 -17250.607,E2 -17250.607} C_VEL
LIN {X 0,Y 305.007,Z 331.707,A -85,B 0,C 180,E1 -17251.459,E2 -17251.459} C_VEL
LIN {X 0,Y 305.227,Z 330.011,A -85,B 0,C 180,E1 -17251.538,E2 -17251.538} C_VEL
LIN {X 0,Y 304.171,Z 330.316,A -85,B 0,C 180,E1 -17251.677,E2 -17251.677} C_VEL
LIN {X 0,Y 300.299,Z 333.791,A -85,B 0,C 180,E1 -17252.036,E2 -17252.036} C_VEL
LIN {X 0,Y 297.215,Z 335.303,A -85,B 0,C 180,E1 -17252.414,E2 -17252.414} C_VEL
LIN {X 0,Y 293.719,Z 335.638,A -85,B 0,C 180,E1 -17252.959,E2 -17252.959} C_VEL
LIN {X 0,Y 291.366,Z 337.688,A -85,B 0,C 180,E1 -17253.186,E2 -17253.186} C_VEL
LIN {X 0,Y 287.022,Z 338.759,A -85,B 0,C 180,E1 -17253.848,E2 -17253.848} C_VEL
LIN {X 0,Y 285.853,Z 336.827,A -85,B 0,C 180,E1 -17254.223,E2 -17254.223} C_VEL
LIN {X 0,Y 285.798,Z 336.439,A -85,B 0,C 180,E1 -17254.266,E2 -17254.266} C_VEL
LIN {X 0,Y 283.937,Z 352.816,A -85,B 0,C 180,E1 -17256.089,E2 -17256.089} C_VEL
LIN {X 0,Y 282.323,Z 366.015,A -85,B 0,C 180,E1 -17257.882,E2 -17257.882} C_VEL
LIN {X 0,Y 280.733,Z 378.218,A -85,B 0,C 180,E1 -17259.865,E2 -17259.865} C_VEL
LIN {X 0,Y 279.338,Z 389.483,A -85,B 0,C 180,E1 -17262.048,E2 -17262.048} C_VEL
LIN {X 0,Y 278.139,Z 399.018,A -85,B 0,C 180,E1 -17264.238,E2 -17264.238} C_VEL
LIN {X 0,Y 277.2,Z 408.385,A -85,B 0,C 180,E1 -17266.809,E2 -17266.809} C_VEL
LIN {X 0,Y 276.456,Z 415.141,A -85,B 0,C 180,E1 -17269.008,E2 -17269.008} C_VEL
LIN {X 0,Y 275.898,Z 422.528,A -85,B 0,C 180,E1 -17271.946,E2 -17271.946} C_VEL
LIN {X 0,Y 275.571,Z 428.295,A -85,B 0,C 180,E1 -17274.878,E2 -17274.878} C_VEL
LIN {X 0,Y 275.55,Z 431.657,A -85,B 0,C 180,E1 -17277.076,E2 -17277.076} C_VEL
LIN {X 0,Y 275.498,Z 434.957,A -85,B 0,C 180,E1 -17280,E2 -17280} C_VEL
LIN {X 0,Y 275.812,Z 436.99,A -85,B 0,C 180,E1 -17282.921,E2 -17282.921} C_VEL
LIN {X 0,Y 276.243,Z 437.823,A -85,B 0,C 180,E1 -17285.84,E2 -17285.84} C_VEL
LIN {X 0,Y 277.227,Z 437.46,A -85,B 0,C 180,E1 -17288.749,E2 -17288.749} C_VEL
LIN {X 0,Y 278.59,Z 435.922,A -85,B 0,C 180,E1 -17291.643,E2 -17291.643} C_VEL
LIN {X 0,Y 280.288,Z 433.193,A -85,B 0,C 180,E1 -17294.521,E2 -17294.521} C_VEL
LIN {X 0,Y 282.773,Z 429.231,A -85,B 0,C 180,E1 -17297.352,E2 -17297.352} C_VEL
LIN {X 0,Y 285.851,Z 424.008,A -85,B 0,C 180,E1 -17300.133,E2 -17300.133} C_VEL
LIN {X 0,Y 289.607,Z 417.409,A -85,B 0,C 180,E1 -17302.847,E2 -17302.847} C_VEL
LIN {X 0,Y 293.925,Z 409.329,A -85,B 0,C 180,E1 -17305.492,E2 -17305.492} C_VEL
LIN {X 0,Y 298.944,Z 399.535,A -85,B 0,C 180,E1 -17308.046,E2 -17308.046} C_VEL
LIN {X 0,Y 303.904,Z 389.332,A -85,B 0,C 180,E1 -17310.197,E2 -17310.197} C_VEL
LIN {X 0,Y 308.923,Z 378.081,A -85,B 0,C 180,E1 -17312.183,E2 -17312.183} C_VEL
LIN {X 0,Y 314.728,Z 364.247,A -85,B 0,C 180,E1 -17314.128,E2 -17314.128} C_VEL
LIN {X 0,Y 320.098,Z 349.972,A -85,B 0,C 180,E1 -17315.772,E2 -17315.772} C_VEL
LIN {X 0,Y 324.971,Z 335.688,A -85,B 0,C 180,E1 -17317.073,E2 -17317.073} C_VEL
LIN {X 0,Y 329.598,Z 320.196,A -85,B 0,C 180,E1 -17318.196,E2 -17318.196} C_VEL
LIN {X 0,Y 333.781,Z 303.443,A -85,B 0,C 180,E1 -17319.125,E2 -17319.125} C_VEL
LIN {X 0,Y 350.524,Z 228.791,A -85,B 0,C 180,E1 -17322.076,E2 -17322.076} C_VEL
LIN {X 0,Y 350.36,Z 228.428,A -85,B 0,C 180,E1 -17322.452,E2 -17322.452} C_VEL
LIN {X 0,Y 349.672,Z 228.832,A -85,B 0,C 180,E1 -17324.432,E2 -17324.432} C_VEL
LIN {X 0,Y 349.671,Z 230.966,A -85,B 0,C 180,E1 -17326.249,E2 -17326.249} C_VEL
LIN {X 0,Y 349.761,Z 233.401,A -85,B 0,C 180,E1 -17327.226,E2 -17327.226} C_VEL
LIN {X 0,Y 331.1,Z 318.495,A -85,B 0,C 180,E1 -17330.595,E2 -17330.595} C_VEL
LIN {X 0,Y 326.134,Z 336.585,A -85,B 0,C 180,E1 -17331.52,E2 -17331.52} C_VEL
LIN {X 0,Y 320.409,Z 354.162,A -85,B 0,C 180,E1 -17332.703,E2 -17332.703} C_VEL
LIN {X 0,Y 314.577,Z 370.133,A -85,B 0,C 180,E1 -17334.094,E2 -17334.094} C_VEL
LIN {X 0,Y 308.821,Z 384.75,A -85,B 0,C 180,E1 -17335.719,E2 -17335.719} C_VEL
LIN {X 0,Y 303.495,Z 397.32,A -85,B 0,C 180,E1 -17337.425,E2 -17337.425} C_VEL
LIN {X 0,Y 297.983,Z 409.966,A -85,B 0,C 180,E1 -17339.53,E2 -17339.53} C_VEL
LIN {X 0,Y 292.461,Z 422.218,A -85,B 0,C 180,E1 -17342.057,E2 -17342.057} C_VEL
LIN {X 0,Y 288.284,Z 431.578,A -85,B 0,C 180,E1 -17344.423,E2 -17344.423} C_VEL
LIN {X 0,Y 284.367,Z 440.302,A -85,B 0,C 180,E1 -17347.092,E2 -17347.092} C_VEL
LIN {X 0,Y 280.833,Z 448.533,A -85,B 0,C 180,E1 -17350.254,E2 -17350.254} C_VEL
LIN {X 0,Y 276.627,Z 461.862,A -85,B 0,C 180,E1 -17356.782,E2 -17356.782} C_VEL
LIN {X 0,Y 275.741,Z 466.452,A -85,B 0,C 180,E1 -17359.723,E2 -17359.723} C_VEL
LIN {X 0,Y 275.367,Z 469.745,A -85,B 0,C 180,E1 -17362.668,E2 -17362.668} C_VEL
LIN {X 0,Y 275.226,Z 471.787,A -85,B 0,C 180,E1 -17365.606,E2 -17365.606} C_VEL
LIN {X 0,Y 275.276,Z 472.641,A -85,B 0,C 180,E1 -17368.537,E2 -17368.537} C_VEL
LIN {X 0,Y 275.278,Z 472.305,A -85,B 0,C 180,E1 -17371.463,E2 -17371.463} C_VEL
LIN {X 0,Y 275.241,Z 470.765,A -85,B 0,C 180,E1 -17374.393,E2 -17374.393} C_VEL
LIN {X 0,Y 275.369,Z 467.982,A -85,B 0,C 180,E1 -17377.332,E2 -17377.332} C_VEL
LIN {X 0,Y 275.673,Z 463.883,A -85,B 0,C 180,E1 -17380.28,E2 -17380.28} C_VEL
LIN {X 0,Y 276.49,Z 458.531,A -85,B 0,C 180,E1 -17383.225,E2 -17383.225} C_VEL
LIN {X 0,Y 277.829,Z 454.166,A -85,B 0,C 180,E1 -17386.156,E2 -17386.156} C_VEL
LIN {X 0,Y 280.056,Z 448.569,A -85,B 0,C 180,E1 -17389.04,E2 -17389.04} C_VEL
LIN {X 0,Y 282.964,Z 441.612,A -85,B 0,C 180,E1 -17391.873,E2 -17391.873} C_VEL
LIN {X 0,Y 286.564,Z 433.191,A -85,B 0,C 180,E1 -17394.641,E2 -17394.641} C_VEL
LIN {X 0,Y 290.455,Z 424.534,A -85,B 0,C 180,E1 -17396.98,E2 -17396.98} C_VEL
LIN {X 0,Y 295.744,Z 412.839,A -85,B 0,C 180,E1 -17399.544,E2 -17399.544} C_VEL
LIN {X 0,Y 300.995,Z 400.82,A -85,B 0,C 180,E1 -17401.692,E2 -17401.692} C_VEL
LIN {X 0,Y 306.502,Z 387.767,A -85,B 0,C 180,E1 -17403.585,E2 -17403.585} C_VEL
LIN {X 0,Y 312.079,Z 373.756,A -85,B 0,C 180,E1 -17405.245,E2 -17405.245} C_VEL
LIN {X 0,Y 317.772,Z 358.56,A -85,B 0,C 180,E1 -17406.666,E2 -17406.666} C_VEL
LIN {X 0,Y 323.32,Z 341.831,A -85,B 0,C 180,E1 -17407.884,E2 -17407.884} C_VEL
LIN {X 0,Y 328.091,Z 325.432,A -85,B 0,C 180,E1 -17408.797,E2 -17408.797} C_VEL
LIN {X 0,Y 332.693,Z 305.807,A -85,B 0,C 180,E1 -17409.67,E2 -17409.67} C_VEL
LIN {X 0,Y 349.204,Z 229.573,A -85,B 0,C 180,E1 -17412.651,E2 -17412.651} C_VEL
LIN {X 0,Y 350.442,Z 224.139,A -85,B 0,C 180,E1 -17412.88,E2 -17412.88} C_VEL
LIN {X 0,Y 350.229,Z 223.205,A -85,B 0,C 180,E1 -17413.493,E2 -17413.493} C_VEL
LIN {X 0,Y 349.811,Z 222.328,A -85,B 0,C 180,E1 -17415.318,E2 -17415.318} C_VEL
LIN {X 0,Y 350.145,Z 222.733,A -85,B 0,C 180,E1 -17417.208,E2 -17417.208} C_VEL
LIN {X 0,Y 350.433,Z 223.37,A -85,B 0,C 180,E1 -17417.935,E2 -17417.935} C_VEL
LIN {X 0,Y 334.738,Z 293.919,A -85,B 0,C 180,E1 -17420.669,E2 -17420.669} C_VEL
LIN {X 0,Y 330.921,Z 311.331,A -85,B 0,C 180,E1 -17421.499,E2 -17421.499} C_VEL
LIN {X 0,Y 326.984,Z 325.978,A -85,B 0,C 180,E1 -17422.42,E2 -17422.42} C_VEL
LIN {X 0,Y 322.546,Z 340.526,A -85,B 0,C 180,E1 -17423.577,E2 -17423.577} C_VEL
LIN {X 0,Y 317.375,Z 355.237,A -85,B 0,C 180,E1 -17425.042,E2 -17425.042} C_VEL
LIN {X 0,Y 312.163,Z 368.667,A -85,B 0,C 180,E1 -17426.717,E2 -17426.717} C_VEL
LIN {X 0,Y 307.69,Z 379.34,A -85,B 0,C 180,E1 -17428.309,E2 -17428.309} C_VEL
LIN {X 0,Y 302.419,Z 390.99,A -85,B 0,C 180,E1 -17430.407,E2 -17430.407} C_VEL
LIN {X 0,Y 297.605,Z 400.875,A -85,B 0,C 180,E1 -17432.581,E2 -17432.581} C_VEL
LIN {X 0,Y 293.31,Z 409.291,A -85,B 0,C 180,E1 -17434.83,E2 -17434.83} C_VEL
LIN {X 0,Y 288.832,Z 417.874,A -85,B 0,C 180,E1 -17437.72,E2 -17437.72} C_VEL
LIN {X 0,Y 285.061,Z 424.54,A -85,B 0,C 180,E1 -17440.56,E2 -17440.56} C_VEL
LIN {X 0,Y 282.064,Z 429.541,A -85,B 0,C 180,E1 -17443.35,E2 -17443.35} C_VEL
LIN {X 0,Y 280.3,Z 432.466,A -85,B 0,C 180,E1 -17445.48,E2 -17445.48} C_VEL
LIN {X 0,Y 278.593,Z 435.24,A -85,B 0,C 180,E1 -17448.357,E2 -17448.357} C_VEL
LIN {X 0,Y 277.15,Z 436.85,A -85,B 0,C 180,E1 -17451.249,E2 -17451.249} C_VEL
LIN {X 0,Y 276.21,Z 437.279,A -85,B 0,C 180,E1 -17454.159,E2 -17454.159} C_VEL
LIN {X 0,Y 275.779,Z 436.505,A -85,B 0,C 180,E1 -17457.079,E2 -17457.079} C_VEL
LIN {X 0,Y 275.489,Z 434.524,A -85,B 0,C 180,E1 -17460,E2 -17460} C_VEL
LIN {X 0,Y 275.519,Z 431.267,A -85,B 0,C 180,E1 -17462.925,E2 -17462.925} C_VEL
LIN {X 0,Y 275.619,Z 426.64,A -85,B 0,C 180,E1 -17465.855,E2 -17465.855} C_VEL
LIN {X 0,Y 275.902,Z 422.211,A -85,B 0,C 180,E1 -17468.054,E2 -17468.054} C_VEL
LIN {X 0,Y 276.41,Z 414.871,A -85,B 0,C 180,E1 -17470.994,E2 -17470.994} C_VEL
LIN {X 0,Y 277.273,Z 406.932,A -85,B 0,C 180,E1 -17473.56,E2 -17473.56} C_VEL
LIN {X 0,Y 278.2,Z 397.338,A -85,B 0,C 180,E1 -17476.135,E2 -17476.135} C_VEL
LIN {X 0,Y 279.679,Z 385.747,A -85,B 0,C 180,E1 -17478.687,E2 -17478.687} C_VEL
LIN {X 0,Y 281.22,Z 373.846,A -85,B 0,C 180,E1 -17480.863,E2 -17480.863} C_VEL
LIN {X 0,Y 282.773,Z 360.553,A -85,B 0,C 180,E1 -17482.891,E2 -17482.891} C_VEL
LIN {X 0,Y 284.366,Z 348.225,A -85,B 0,C 180,E1 -17484.455,E2 -17484.455} C_VEL
LIN {X 0,Y 286.017,Z 332.959,A -85,B 0,C 180,E1 -17486.055,E2 -17486.055} C_VEL
LIN {X 0,Y 287.554,Z 317.126,A -85,B 0,C 180,E1 -17487.374,E2 -17487.374} C_VEL
LIN {X 0,Y 288.798,Z 300.622,A -85,B 0,C 180,E1 -17488.429,E2 -17488.429} C_VEL
LIN {X 0,Y 289.843,Z 283.205,A -85,B 0,C 180,E1 -17489.216,E2 -17489.216} C_VEL
LIN {X 0,Y 295.725,Z 180.459,A -85,B 0,C 180,E1 -17492.896,E2 -17492.896} C_VEL
LIN {X 0,Y 277.346,Z 136.84,A -85,B 0,C 180,E1 -17496.212,E2 -17496.212} C_VEL
LIN {X 0,Y 277.29,Z 136.569,A -85,B 0,C 180,E1 -17496.253,E2 -17496.253} C_VEL
LIN {X 0,Y 277.199,Z 136.581,A -85,B 0,C 180,E1 -17500.482,E2 -17500.482} C_VEL
LIN {X 0,Y 277.193,Z 136.579,A -85,B 0,C 180,E1 -17503.202,E2 -17503.202} C_VEL
LIN {X 0,Y 277.193,Z 136.546,A -85,B 0,C 180,E1 -17507.331,E2 -17507.331} C_VEL
LIN {X 0,Y 277.254,Z 136.57,A -85,B 0,C 180,E1 -17511.796,E2 -17511.796} C_VEL
LIN {X 0,Y 277.28,Z 136.541,A -85,B 0,C 180,E1 -17514.341,E2 -17514.341} C_VEL
LIN {X 0,Y 277.242,Z 136.575,A -85,B 0,C 180,E1 -17517.836,E2 -17517.836} C_VEL
LIN {X 0,Y 277.241,Z 136.556,A -85,B 0,C 180,E1 -17521.207,E2 -17521.207} C_VEL
LIN {X 0,Y 277.235,Z 136.569,A -85,B 0,C 180,E1 -17524.472,E2 -17524.472} C_VEL
LIN {X 0,Y 277.25,Z 136.574,A -85,B 0,C 180,E1 -17527.652,E2 -17527.652} C_VEL
LIN {X 0,Y 277.282,Z 136.559,A -85,B 0,C 180,E1 -17530.762,E2 -17530.762} C_VEL
LIN {X 0,Y 277.328,Z 136.608,A -85,B 0,C 180,E1 -17533.53,E2 -17533.53} C_VEL
LIN {X 0,Y 280.695,Z 145.86,A -85,B 0,C 180,E1 -17536.018,E2 -17536.018} C_VEL
LIN {X 0,Y 291.86,Z 166.243,A -85,B 0,C 180,E1 -17538.302,E2 -17538.302} C_VEL
LIN {X 0,Y 298.525,Z 180.382,A -85,B 0,C 180,E1 -17539.622,E2 -17539.622} C_VEL
LIN {X 0,Y 304.992,Z 195.262,A -85,B 0,C 180,E1 -17540.875,E2 -17540.875} C_VEL
LIN {X 0,Y 301.512,Z 283.06,A -85,B 0,C 180,E1 -17542.971,E2 -17542.971} C_VEL
LIN {X 0,Y 300.215,Z 313.802,A -85,B 0,C 180,E1 -17543.742,E2 -17543.742} C_VEL
LIN {X 0,Y 298.952,Z 329.173,A -85,B 0,C 180,E1 -17544.35,E2 -17544.35} C_VEL
LIN {X 0,Y 297.352,Z 344.576,A -85,B 0,C 180,E1 -17545.255,E2 -17545.255} C_VEL
LIN {X 0,Y 295.252,Z 359.419,A -85,B 0,C 180,E1 -17546.409,E2 -17546.409} C_VEL
LIN {X 0,Y 293.021,Z 373.006,A -85,B 0,C 180,E1 -17547.766,E2 -17547.766} C_VEL
LIN {X 0,Y 290.597,Z 385.531,A -85,B 0,C 180,E1 -17549.307,E2 -17549.307} C_VEL
LIN {X 0,Y 287.973,Z 398.068,A -85,B 0,C 180,E1 -17551.201,E2 -17551.201} C_VEL
LIN {X 0,Y 285.537,Z 408.845,A -85,B 0,C 180,E1 -17553.175,E2 -17553.175} C_VEL
LIN {X 0,Y 283.194,Z 418.684,A -85,B 0,C 180,E1 -17555.34,E2 -17555.34} C_VEL
LIN {X 0,Y 280.87,Z 428.294,A -85,B 0,C 180,E1 -17557.91,E2 -17557.91} C_VEL
LIN {X 0,Y 278.931,Z 436.687,A -85,B 0,C 180,E1 -17560.685,E2 -17560.685} C_VEL
LIN {X 0,Y 277.581,Z 442.784,A -85,B 0,C 180,E1 -17563.172,E2 -17563.172} C_VEL
LIN {X 0,Y 276.407,Z 448.73,A -85,B 0,C 180,E1 -17566.242,E2 -17566.242} C_VEL
LIN {X 0,Y 275.583,Z 453.213,A -85,B 0,C 180,E1 -17569.362,E2 -17569.362} C_VEL
LIN {X 0,Y 275.089,Z 456.295,A -85,B 0,C 180,E1 -17572.533,E2 -17572.533} C_VEL
LIN {X 0,Y 274.906,Z 457.994,A -85,B 0,C 180,E1 -17575.76,E2 -17575.76} C_VEL
LIN {X 0,Y 274.949,Z 458.288,A -85,B 0,C 180,E1 -17579.056,E2 -17579.056} C_VEL
LIN {X 0,Y 275.248,Z 457.098,A -85,B 0,C 180,E1 -17582.425,E2 -17582.425} C_VEL
LIN {X 0,Y 275.859,Z 454.767,A -85,B 0,C 180,E1 -17585.386,E2 -17585.386} C_VEL
LIN {X 0,Y 276.682,Z 451.617,A -85,B 0,C 180,E1 -17588.053,E2 -17588.053} C_VEL
LIN {X 0,Y 277.992,Z 446.709,A -85,B 0,C 180,E1 -17591.095,E2 -17591.095} C_VEL
LIN {X 0,Y 279.641,Z 441.015,A -85,B 0,C 180,E1 -17593.806,E2 -17593.806} C_VEL
LIN {X 0,Y 281.654,Z 434.37,A -85,B 0,C 180,E1 -17596.355,E2 -17596.355} C_VEL
LIN {X 0,Y 284.261,Z 426.023,A -85,B 0,C 180,E1 -17598.945,E2 -17598.945} C_VEL
LIN {X 0,Y 287.305,Z 415.791,A -85,B 0,C 180,E1 -17601.516,E2 -17601.516} C_VEL
LIN {X 0,Y 289.001,Z 409.88,A -85,B 0,C 180,E1 -17602.778,E2 -17602.778} C_VEL
LIN {X 0,Y 289.562,Z 405.883,A -85,B 0,C 180,E1 -17603.633,E2 -17603.633} C_VEL
LIN {X 0,Y 288.914,Z 399.36,A -85,B 0,C 180,E1 -17605.116,E2 -17605.116} C_VEL
LIN {X 0,Y 288.346,Z 392.49,A -85,B 0,C 180,E1 -17606.526,E2 -17606.526} C_VEL
LIN {X 0,Y 288.991,Z 387.911,A -85,B 0,C 180,E1 -17607.251,E2 -17607.251} C_VEL
LIN {X 0,Y 291.852,Z 376.181,A -85,B 0,C 180,E1 -17608.745,E2 -17608.745} C_VEL
LIN {X 0,Y 294.847,Z 361.912,A -85,B 0,C 180,E1 -17610.206,E2 -17610.206} C_VEL
LIN {X 0,Y 297.343,Z 347.761,A -85,B 0,C 180,E1 -17611.337,E2 -17611.337} C_VEL
LIN {X 0,Y 298.13,Z 342.521,A -85,B 0,C 180,E1 -17611.694,E2 -17611.694} C_VEL
LIN {X 0,Y 297.702,Z 341.718,A -85,B 0,C 180,E1 -17611.826,E2 -17611.826} C_VEL
LIN {X 0,Y 293.481,Z 343.074,A -85,B 0,C 180,E1 -17612.38,E2 -17612.38} C_VEL
LIN {X 0,Y 290.966,Z 344.296,A -85,B 0,C 180,E1 -17612.682,E2 -17612.682} C_VEL
LIN {X 0,Y 284.736,Z 345.67,A -85,B 0,C 180,E1 -17613.622,E2 -17613.622} C_VEL
LIN {X 0,Y 281.436,Z 347.55,A -85,B 0,C 180,E1 -17614.026,E2 -17614.026} C_VEL
LIN {X 0,Y 278.592,Z 347.069,A -85,B 0,C 180,E1 -17614.604,E2 -17614.604} C_VEL
LIN {X 0,Y 277.864,Z 345.41,A -85,B 0,C 180,E1 -17614.934,E2 -17614.934} C_VEL
LIN {X 0,Y 276.004,Z 360.364,A -85,B 0,C 180,E1 -17616.825,E2 -17616.825} C_VEL
LIN {X 0,Y 274.44,Z 373.158,A -85,B 0,C 180,E1 -17618.794,E2 -17618.794} C_VEL
LIN {X 0,Y 272.95,Z 384.322,A -85,B 0,C 180,E1 -17620.834,E2 -17620.834} C_VEL
LIN {X 0,Y 271.602,Z 394.862,A -85,B 0,C 180,E1 -17623.114,E2 -17623.114} C_VEL
LIN {X 0,Y 270.509,Z 404.897,A -85,B 0,C 180,E1 -17625.71,E2 -17625.71} C_VEL
LIN {X 0,Y 269.52,Z 413.317,A -85,B 0,C 180,E1 -17628.34,E2 -17628.34} C_VEL
LIN {X 0,Y 268.977,Z 420.289,A -85,B 0,C 180,E1 -17630.98,E2 -17630.98} C_VEL
LIN {X 0,Y 268.56,Z 426.678,A -85,B 0,C 180,E1 -17633.991,E2 -17633.991} C_VEL
LIN {X 0,Y 268.476,Z 431.544,A -85,B 0,C 180,E1 -17636.998,E2 -17636.998} C_VEL
LIN {X 0,Y 268.413,Z 435.048,A -85,B 0,C 180,E1 -17640,E2 -17640} C_VEL
LIN {X 0,Y 268.734,Z 437.285,A -85,B 0,C 180,E1 -17642.998,E2 -17642.998} C_VEL
LIN {X 0,Y 269.215,Z 438.329,A -85,B 0,C 180,E1 -17645.993,E2 -17645.993} C_VEL
LIN {X 0,Y 270.243,Z 438.141,A -85,B 0,C 180,E1 -17648.977,E2 -17648.977} C_VEL
LIN {X 0,Y 271.673,Z 436.784,A -85,B 0,C 180,E1 -17651.944,E2 -17651.944} C_VEL
LIN {X 0,Y 273.5,Z 434.299,A -85,B 0,C 180,E1 -17654.89,E2 -17654.89} C_VEL
LIN {X 0,Y 276.135,Z 430.605,A -85,B 0,C 180,E1 -17657.783,E2 -17657.783} C_VEL
LIN {X 0,Y 279.383,Z 425.682,A -85,B 0,C 180,E1 -17660.62,E2 -17660.62} C_VEL
LIN {X 0,Y 283.448,Z 419.237,A -85,B 0,C 180,E1 -17663.451,E2 -17663.451} C_VEL
LIN {X 0,Y 288.487,Z 410.635,A -85,B 0,C 180,E1 -17666.397,E2 -17666.397} C_VEL
LIN {X 0,Y 293.854,Z 401.075,A -85,B 0,C 180,E1 -17668.967,E2 -17668.967} C_VEL
LIN {X 0,Y 299.081,Z 391.177,A -85,B 0,C 180,E1 -17671.129,E2 -17671.129} C_VEL
LIN {X 0,Y 304.703,Z 379.64,A -85,B 0,C 180,E1 -17673.216,E2 -17673.216} C_VEL
LIN {X 0,Y 310.75,Z 366.463,A -85,B 0,C 180,E1 -17675.122,E2 -17675.122} C_VEL
LIN {X 0,Y 316.63,Z 352.092,A -85,B 0,C 180,E1 -17676.819,E2 -17676.819} C_VEL
LIN {X 0,Y 321.762,Z 338.293,A -85,B 0,C 180,E1 -17678.1,E2 -17678.1} C_VEL
LIN {X 0,Y 326.752,Z 322.988,A -85,B 0,C 180,E1 -17679.239,E2 -17679.239} C_VEL
LIN {X 0,Y 331.204,Z 306.915,A -85,B 0,C 180,E1 -17680.167,E2 -17680.167} C_VEL
LIN {X 0,Y 336.97,Z 281.944,A -85,B 0,C 180,E1 -17681.218,E2 -17681.218} C_VEL
LIN {X 0,Y 348.232,Z 235.294,A -85,B 0,C 180,E1 -17683.028,E2 -17683.028} C_VEL
LIN {X 0,Y 347.791,Z 235.936,A -85,B 0,C 180,E1 -17684.703,E2 -17684.703} C_VEL
LIN {X 0,Y 347.717,Z 237.983,A -85,B 0,C 180,E1 -17686.122,E2 -17686.122} C_VEL
LIN {X 0,Y 347.684,Z 238.397,A -85,B 0,C 180,E1 -17686.246,E2 -17686.246} C_VEL
LIN {X 0,Y 329.481,Z 316.557,A -85,B 0,C 180,E1 -17689.314,E2 -17689.314} C_VEL
LIN {X 0,Y 324.16,Z 335.027,A -85,B 0,C 180,E1 -17690.239,E2 -17690.239} C_VEL
LIN {X 0,Y 318.115,Z 352.494,A -85,B 0,C 180,E1 -17691.383,E2 -17691.383} C_VEL
LIN {X 0,Y 311.927,Z 368.376,A -85,B 0,C 180,E1 -17692.734,E2 -17692.734} C_VEL
LIN {X 0,Y 306.234,Z 381.822,A -85,B 0,C 180,E1 -17694.182,E2 -17694.182} C_VEL
LIN {X 0,Y 299.647,Z 396.5,A -85,B 0,C 180,E1 -17696.149,E2 -17696.149} C_VEL
LIN {X 0,Y 293.709,Z 409.016,A -85,B 0,C 180,E1 -17698.236,E2 -17698.236} C_VEL
LIN {X 0,Y 287.787,Z 421.194,A -85,B 0,C 180,E1 -17700.763,E2 -17700.763} C_VEL
LIN {X 0,Y 282.644,Z 431.519,A -85,B 0,C 180,E1 -17703.412,E2 -17703.412} C_VEL
LIN {X 0,Y 278.351,Z 440.237,A -85,B 0,C 180,E1 -17706.173,E2 -17706.173} C_VEL
LIN {X 0,Y 274.919,Z 447.519,A -85,B 0,C 180,E1 -17709.029,E2 -17709.029} C_VEL
LIN {X 0,Y 272.157,Z 453.451,A -85,B 0,C 180,E1 -17711.948,E2 -17711.948} C_VEL
LIN {X 0,Y 270.902,Z 456.496,A -85,B 0,C 180,E1 -17713.716,E2 -17713.716} C_VEL
LIN {X 0,Y 269.671,Z 461.807,A -85,B 0,C 180,E1 -17716.435,E2 -17716.435} C_VEL
LIN {X 0,Y 268.714,Z 466.359,A -85,B 0,C 180,E1 -17719.451,E2 -17719.451} C_VEL
LIN {X 0,Y 268.286,Z 469.627,A -85,B 0,C 180,E1 -17722.474,E2 -17722.474} C_VEL
LIN {X 0,Y 268.141,Z 471.644,A -85,B 0,C 180,E1 -17725.49,E2 -17725.49} C_VEL
LIN {X 0,Y 268.201,Z 472.463,A -85,B 0,C 180,E1 -17728.498,E2 -17728.498} C_VEL
LIN {X 0,Y 268.204,Z 472.094,A -85,B 0,C 180,E1 -17731.502,E2 -17731.502} C_VEL
LIN {X 0,Y 268.156,Z 470.518,A -85,B 0,C 180,E1 -17734.51,E2 -17734.51} C_VEL
LIN {X 0,Y 268.286,Z 467.698,A -85,B 0,C 180,E1 -17737.526,E2 -17737.526} C_VEL
LIN {X 0,Y 268.626,Z 463.558,A -85,B 0,C 180,E1 -17740.553,E2 -17740.553} C_VEL
LIN {X 0,Y 269.233,Z 459.535,A -85,B 0,C 180,E1 -17742.82,E2 -17742.82} C_VEL
LIN {X 0,Y 270.972,Z 454.464,A -85,B 0,C 180,E1 -17746.577,E2 -17746.577} C_VEL
LIN {X 0,Y 273.34,Z 449.122,A -85,B 0,C 180,E1 -17749.527,E2 -17749.527} C_VEL
LIN {X 0,Y 276.435,Z 442.477,A -85,B 0,C 180,E1 -17752.418,E2 -17752.418} C_VEL
LIN {X 0,Y 280.23,Z 434.46,A -85,B 0,C 180,E1 -17755.236,E2 -17755.236} C_VEL
LIN {X 0,Y 284.962,Z 424.863,A -85,B 0,C 180,E1 -17757.943,E2 -17757.943} C_VEL
LIN {X 0,Y 290.586,Z 413.441,A -85,B 0,C 180,E1 -17760.524,E2 -17760.524} C_VEL
LIN {X 0,Y 296.133,Z 401.751,A -85,B 0,C 180,E1 -17762.678,E2 -17762.678} C_VEL
LIN {X 0,Y 301.926,Z 389.175,A -85,B 0,C 180,E1 -17764.568,E2 -17764.568} C_VEL
LIN {X 0,Y 308.258,Z 374.509,A -85,B 0,C 180,E1 -17766.354,E2 -17766.354} C_VEL
LIN {X 0,Y 314.789,Z 358.316,A -85,B 0,C 180,E1 -17767.877,E2 -17767.877} C_VEL
LIN {X 0,Y 320,Z 343.79,A -85,B 0,C 180,E1 -17768.953,E2 -17768.953} C_VEL
LIN {X 0,Y 325.277,Z 327.256,A -85,B 0,C 180,E1 -17769.899,E2 -17769.899} C_VEL
LIN {X 0,Y 330.549,Z 306.712,A -85,B 0,C 180,E1 -17770.828,E2 -17770.828} C_VEL
LIN {X 0,Y 348.2,Z 230.171,A -85,B 0,C 180,E1 -17773.813,E2 -17773.813} C_VEL
LIN {X 0,Y 348.247,Z 229.811,A -85,B 0,C 180,E1 -17773.903,E2 -17773.903} C_VEL
LIN {X 0,Y 348.021,Z 229.245,A -85,B 0,C 180,E1 -17775.025,E2 -17775.025} C_VEL
LIN {X 0,Y 348.233,Z 229.447,A -85,B 0,C 180,E1 -17776.984,E2 -17776.984} C_VEL
LIN {X 0,Y 331.014,Z 302.986,A -85,B 0,C 180,E1 -17779.863,E2 -17779.863} C_VEL
LIN {X 0,Y 327.084,Z 318.221,A -85,B 0,C 180,E1 -17780.678,E2 -17780.678} C_VEL
LIN {X 0,Y 321.767,Z 335.491,A -85,B 0,C 180,E1 -17781.901,E2 -17781.901} C_VEL
LIN {X 0,Y 316.181,Z 350.888,A -85,B 0,C 180,E1 -17783.319,E2 -17783.319} C_VEL
LIN {X 0,Y 311.23,Z 363.201,A -85,B 0,C 180,E1 -17784.724,E2 -17784.724} C_VEL
LIN {X 0,Y 305.628,Z 376.016,A -85,B 0,C 180,E1 -17786.504,E2 -17786.504} C_VEL
LIN {X 0,Y 299.87,Z 388.13,A -85,B 0,C 180,E1 -17788.57,E2 -17788.57} C_VEL
LIN {X 0,Y 293.805,Z 399.824,A -85,B 0,C 180,E1 -17791.028,E2 -17791.028} C_VEL
LIN {X 0,Y 288.462,Z 409.473,A -85,B 0,C 180,E1 -17793.6,E2 -17793.6} C_VEL
LIN {X 0,Y 284.357,Z 416.742,A -85,B 0,C 180,E1 -17796.011,E2 -17796.011} C_VEL
LIN {X 0,Y 280.397,Z 423.292,A -85,B 0,C 180,E1 -17798.689,E2 -17798.689} C_VEL
LIN {X 0,Y 276.839,Z 428.693,A -85,B 0,C 180,E1 -17801.499,E2 -17801.499} C_VEL
LIN {X 0,Y 274.795,Z 431.812,A -85,B 0,C 180,E1 -17803.661,E2 -17803.661} C_VEL
LIN {X 0,Y 272.55,Z 434.975,A -85,B 0,C 180,E1 -17806.581,E2 -17806.581} C_VEL
LIN {X 0,Y 270.879,Z 436.972,A -85,B 0,C 180,E1 -17809.537,E2 -17809.537} C_VEL
LIN {X 0,Y 269.567,Z 437.814,A -85,B 0,C 180,E1 -17812.51,E2 -17812.51} C_VEL
LIN {X 0,Y 268.892,Z 437.426,A -85,B 0,C 180,E1 -17815.503,E2 -17815.503} C_VEL
LIN {X 0,Y 268.497,Z 435.85,A -85,B 0,C 180,E1 -17818.501,E2 -17818.501} C_VEL
LIN {X 0,Y 268.373,Z 433.036,A -85,B 0,C 180,E1 -17821.501,E2 -17821.501} C_VEL
LIN {X 0,Y 268.449,Z 428.905,A -85,B 0,C 180,E1 -17824.505,E2 -17824.505} C_VEL
LIN {X 0,Y 268.744,Z 423.338,A -85,B 0,C 180,E1 -17827.514,E2 -17827.514} C_VEL
LIN {X 0,Y 269.07,Z 418.143,A -85,B 0,C 180,E1 -17829.775,E2 -17829.775} C_VEL
LIN {X 0,Y 269.716,Z 410.819,A -85,B 0,C 180,E1 -17832.414,E2 -17832.414} C_VEL
LIN {X 0,Y 270.693,Z 401.936,A -85,B 0,C 180,E1 -17835.049,E2 -17835.049} C_VEL
LIN {X 0,Y 271.719,Z 392.882,A -85,B 0,C 180,E1 -17837.304,E2 -17837.304} C_VEL
LIN {X 0,Y 273.045,Z 382.22,A -85,B 0,C 180,E1 -17839.549,E2 -17839.549} C_VEL
LIN {X 0,Y 274.723,Z 369.581,A -85,B 0,C 180,E1 -17841.774,E2 -17841.774} C_VEL
LIN {X 0,Y 276.435,Z 355.971,A -85,B 0,C 180,E1 -17843.758,E2 -17843.758} C_VEL
LIN {X 0,Y 277.903,Z 343.647,A -85,B 0,C 180,E1 -17845.263,E2 -17845.263} C_VEL
LIN {X 0,Y 279.555,Z 328.137,A -85,B 0,C 180,E1 -17846.805,E2 -17846.805} C_VEL
LIN {X 0,Y 281.059,Z 312.1,A -85,B 0,C 180,E1 -17848.062,E2 -17848.062} C_VEL
LIN {X 0,Y 282.24,Z 295.344,A -85,B 0,C 180,E1 -17849.059,E2 -17849.059} C_VEL
LIN {X 0,Y 283.562,Z 272.877,A -85,B 0,C 180,E1 -17849.972,E2 -17849.972} C_VEL
LIN {X 0,Y 288.918,Z 182.039,A -85,B 0,C 180,E1 -17853.34,E2 -17853.34} C_VEL
LIN {X 0,Y 271.942,Z 142.064,A -85,B 0,C 180,E1 -17856.456,E2 -17856.456} C_VEL
LIN {X 0,Y 270.24,Z 137.458,A -85,B 0,C 180,E1 -17856.817,E2 -17856.817} C_VEL
LIN {X 0,Y 270.147,Z 137.461,A -85,B 0,C 180,E1 -17861.023,E2 -17861.023} C_VEL
LIN {X 0,Y 270.131,Z 137.441,A -85,B 0,C 180,E1 -17864.626,E2 -17864.626} C_VEL
LIN {X 0,Y 270.152,Z 137.423,A -85,B 0,C 180,E1 -17867.438,E2 -17867.438} C_VEL
LIN {X 0,Y 270.21,Z 137.45,A -85,B 0,C 180,E1 -17871.375,E2 -17871.375} C_VEL
LIN {X 0,Y 270.2,Z 137.425,A -85,B 0,C 180,E1 -17875.094,E2 -17875.094} C_VEL
LIN {X 0,Y 270.187,Z 137.443,A -85,B 0,C 180,E1 -17879.137,E2 -17879.137} C_VEL
LIN {X 0,Y 270.224,Z 137.44,A -85,B 0,C 180,E1 -17882.163,E2 -17882.163} C_VEL
LIN {X 0,Y 270.184,Z 137.437,A -85,B 0,C 180,E1 -17885.564,E2 -17885.564} C_VEL
LIN {X 0,Y 270.223,Z 137.436,A -85,B 0,C 180,E1 -17890.238,E2 -17890.238} C_VEL
LIN {X 0,Y 270.281,Z 137.587,A -85,B 0,C 180,E1 -17892.504,E2 -17892.504} C_VEL
LIN {X 0,Y 273.479,Z 146.044,A -85,B 0,C 180,E1 -17894.881,E2 -17894.881} C_VEL
LIN {X 0,Y 283.031,Z 163.185,A -85,B 0,C 180,E1 -17896.941,E2 -17896.941} C_VEL
LIN {X 0,Y 290.544,Z 177.976,A -85,B 0,C 180,E1 -17898.488,E2 -17898.488} C_VEL
LIN {X 0,Y 299.101,Z 197.473,A -85,B 0,C 180,E1 -17900.205,E2 -17900.205} C_VEL
LIN {X 0,Y 294.093,Z 313.823,A -85,B 0,C 180,E1 -17903.051,E2 -17903.051} C_VEL
LIN {X 0,Y 292.8,Z 329.238,A -85,B 0,C 180,E1 -17903.67,E2 -17903.67} C_VEL
LIN {X 0,Y 291.23,Z 344.029,A -85,B 0,C 180,E1 -17904.545,E2 -17904.545} C_VEL
LIN {X 0,Y 289.059,Z 358.959,A -85,B 0,C 180,E1 -17905.71,E2 -17905.71} C_VEL
LIN {X 0,Y 286.897,Z 371.978,A -85,B 0,C 180,E1 -17907.016,E2 -17907.016} C_VEL
LIN {X 0,Y 284.301,Z 384.758,A -85,B 0,C 180,E1 -17908.583,E2 -17908.583} C_VEL
LIN {X 0,Y 281.705,Z 396.846,A -85,B 0,C 180,E1 -17910.41,E2 -17910.41} C_VEL
LIN {X 0,Y 279.043,Z 408.352,A -85,B 0,C 180,E1 -17912.526,E2 -17912.526} C_VEL
LIN {X 0,Y 276.588,Z 418.302,A -85,B 0,C 180,E1 -17914.737,E2 -17914.737} C_VEL
LIN {X 0,Y 274.129,Z 428.013,A -85,B 0,C 180,E1 -17917.365,E2 -17917.365} C_VEL
LIN {X 0,Y 272.208,Z 436.037,A -85,B 0,C 180,E1 -17920.036,E2 -17920.036} C_VEL
LIN {X 0,Y 270.66,Z 442.66,A -85,B 0,C 180,E1 -17922.751,E2 -17922.751} C_VEL
LIN {X 0,Y 269.414,Z 448.714,A -85,B 0,C 180,E1 -17925.921,E2 -17925.921} C_VEL
LIN {X 0,Y 268.751,Z 452.248,A -85,B 0,C 180,E1 -17928.289,E2 -17928.289} C_VEL
LIN {X 0,Y 268.095,Z 455.751,A -85,B 0,C 180,E1 -17931.531,E2 -17931.531} C_VEL
LIN {X 0,Y 267.91,Z 457.076,A -85,B 0,C 180,E1 -17933.342,E2 -17933.342} C_VEL
LIN {X 0,Y 267.79,Z 458.39,A -85,B 0,C 180,E1 -17936.497,E2 -17936.497} C_VEL
LIN {X 0,Y 267.907,Z 458.374,A -85,B 0,C 180,E1 -17939.896,E2 -17939.896} C_VEL
LIN {X 0,Y 268.291,Z 456.839,A -85,B 0,C 180,E1 -17943.374,E2 -17943.374} C_VEL
LIN {X 0,Y 268.888,Z 454.781,A -85,B 0,C 180,E1 -17945.878,E2 -17945.878} C_VEL
LIN {X 0,Y 269.846,Z 451.446,A -85,B 0,C 180,E1 -17948.687,E2 -17948.687} C_VEL
LIN {X 0,Y 270.96,Z 447.501,A -85,B 0,C 180,E1 -17951.219,E2 -17951.219} C_VEL
LIN {X 0,Y 272.718,Z 441.764,A -85,B 0,C 180,E1 -17954.091,E2 -17954.091} C_VEL
LIN {X 0,Y 274.998,Z 434.678,A -85,B 0,C 180,E1 -17956.893,E2 -17956.893} C_VEL
LIN {X 0,Y 277.614,Z 426.778,A -85,B 0,C 180,E1 -17959.418,E2 -17959.418} C_VEL
LIN {X 0,Y 280.233,Z 418.49,A -85,B 0,C 180,E1 -17961.603,E2 -17961.603} C_VEL
LIN {X 0,Y 283.397,Z 407.982,A -85,B 0,C 180,E1 -17963.907,E2 -17963.907} C_VEL
LIN {X 0,Y 286.892,Z 395.922,A -85,B 0,C 180,E1 -17966.056,E2 -17966.056} C_VEL
LIN {X 0,Y 288.991,Z 387.911,A -85,B 0,C 180,E1 -17967.251,E2 -17967.251} C_VEL
LIN {X 0,Y 289.667,Z 383.254,A -85,B 0,C 180,E1 -17967.956,E2 -17967.956} C_VEL
LIN {X 0,Y 288.603,Z 369.459,A -85,B 0,C 180,E1 -17970.197,E2 -17970.197} C_VEL
LIN {X 0,Y 288.798,Z 364.467,A -85,B 0,C 180,E1 -17970.821,E2 -17970.821} C_VEL
LIN {X 0,Y 289.069,Z 362.724,A -85,B 0,C 180,E1 -17970.994,E2 -17970.994} C_VEL
LIN {X 0,Y 291.092,Z 351.855,A -85,B 0,C 180,E1 -17971.913,E2 -17971.913} C_VEL
LIN {X 0,Y 288.435,Z 351.237,A -85,B 0,C 180,E1 -17972.422,E2 -17972.422} C_VEL
LIN {X 0,Y 283.784,Z 352.593,A -85,B 0,C 180,E1 -17973.069,E2 -17973.069} C_VEL
LIN {X 0,Y 281.68,Z 353.715,A -85,B 0,C 180,E1 -17973.313,E2 -17973.313} C_VEL
LIN {X 0,Y 275.787,Z 354.326,A -85,B 0,C 180,E1 -17974.327,E2 -17974.327} C_VEL
LIN {X 0,Y 271.129,Z 355.291,A -85,B 0,C 180,E1 -17975.127,E2 -17975.127} C_VEL
LIN {X 0,Y 270.039,Z 353.7,A -85,B 0,C 180,E1 -17975.545,E2 -17975.545} C_VEL
LIN {X 0,Y 269.951,Z 353.294,A -85,B 0,C 180,E1 -17975.614,E2 -17975.614} C_VEL
LIN {X 0,Y 268.137,Z 367.549,A -85,B 0,C 180,E1 -17977.663,E2 -17977.663} C_VEL
LIN {X 0,Y 266.507,Z 379.625,A -85,B 0,C 180,E1 -17979.749,E2 -17979.749} C_VEL
LIN {X 0,Y 264.984,Z 391.656,A -85,B 0,C 180,E1 -17982.241,E2 -17982.241} C_VEL
LIN {X 0,Y 263.651,Z 402.438,A -85,B 0,C 180,E1 -17984.935,E2 -17984.935} C_VEL
LIN {X 0,Y 262.776,Z 410.167,A -85,B 0,C 180,E1 -17987.252,E2 -17987.252} C_VEL
LIN {X 0,Y 262.062,Z 417.773,A -85,B 0,C 180,E1 -17989.961,E2 -17989.961} C_VEL
LIN {X 0,Y 261.565,Z 424.803,A -85,B 0,C 180,E1 -17993.055,E2 -17993.055} C_VEL
LIN {X 0,Y 261.378,Z 430.263,A -85,B 0,C 180,E1 -17996.145,E2 -17996.145} C_VEL
LIN {X 0,Y 261.316,Z 433.426,A -85,B 0,C 180,E1 -17998.458,E2 -17998.458} C_VEL
LIN {X 0,Y 261.452,Z 436.495,A -85,B 0,C 180,E1 -18001.54,E2 -18001.54} C_VEL
LIN {X 0,Y 261.872,Z 438.297,A -85,B 0,C 180,E1 -18004.618,E2 -18004.618} C_VEL
LIN {X 0,Y 262.654,Z 438.907,A -85,B 0,C 180,E1 -18007.688,E2 -18007.688} C_VEL
LIN {X 0,Y 263.939,Z 438.36,A -85,B 0,C 180,E1 -18010.742,E2 -18010.742} C_VEL
LIN {X 0,Y 265.75,Z 436.682,A -85,B 0,C 180,E1 -18013.769,E2 -18013.769} C_VEL
LIN {X 0,Y 268.11,Z 433.871,A -85,B 0,C 180,E1 -18016.758,E2 -18016.758} C_VEL
LIN {X 0,Y 271.137,Z 429.855,A -85,B 0,C 180,E1 -18019.692,E2 -18019.692} C_VEL
LIN {X 0,Y 275.055,Z 424.527,A -85,B 0,C 180,E1 -18022.536,E2 -18022.536} C_VEL
LIN {X 0,Y 279.47,Z 417.921,A -85,B 0,C 180,E1 -18025.309,E2 -18025.309} C_VEL
LIN {X 0,Y 283.861,Z 410.96,A -85,B 0,C 180,E1 -18027.66,E2 -18027.66} C_VEL
LIN {X 0,Y 289.64,Z 401.485,A -85,B 0,C 180,E1 -18030.231,E2 -18030.231} C_VEL
LIN {X 0,Y 296.043,Z 390.186,A -85,B 0,C 180,E1 -18032.689,E2 -18032.689} C_VEL
LIN {X 0,Y 301.243,Z 380.286,A -85,B 0,C 180,E1 -18034.454,E2 -18034.454} C_VEL
LIN {X 0,Y 307.875,Z 366.818,A -85,B 0,C 180,E1 -18036.406,E2 -18036.406} C_VEL
LIN {X 0,Y 314.254,Z 352.369,A -85,B 0,C 180,E1 -18038.087,E2 -18038.087} C_VEL
LIN {X 0,Y 319.833,Z 338.326,A -85,B 0,C 180,E1 -18039.382,E2 -18039.382} C_VEL
LIN {X 0,Y 325.513,Z 321.926,A -85,B 0,C 180,E1 -18040.573,E2 -18040.573} C_VEL
LIN {X 0,Y 330.217,Z 305.609,A -85,B 0,C 180,E1 -18041.469,E2 -18041.469} C_VEL
LIN {X 0,Y 346.052,Z 242.49,A -85,B 0,C 180,E1 -18043.928,E2 -18043.928} C_VEL
LIN {X 0,Y 345.938,Z 242.871,A -85,B 0,C 180,E1 -18044.679,E2 -18044.679} C_VEL
LIN {X 0,Y 345.811,Z 243.762,A -85,B 0,C 180,E1 -18045.257,E2 -18045.257} C_VEL
LIN {X 0,Y 328.329,Z 314.712,A -85,B 0,C 180,E1 -18048.016,E2 -18048.016} C_VEL
LIN {X 0,Y 323.08,Z 332.068,A -85,B 0,C 180,E1 -18048.85,E2 -18048.85} C_VEL
LIN {X 0,Y 317.375,Z 348.093,A -85,B 0,C 180,E1 -18049.838,E2 -18049.838} C_VEL
LIN {X 0,Y 311.34,Z 363.033,A -85,B 0,C 180,E1 -18051.006,E2 -18051.006} C_VEL
LIN {X 0,Y 305.119,Z 377.002,A -85,B 0,C 180,E1 -18052.382,E2 -18052.382} C_VEL
LIN {X 0,Y 298.954,Z 390.058,A -85,B 0,C 180,E1 -18054.005,E2 -18054.005} C_VEL
LIN {X 0,Y 292.315,Z 403.226,A -85,B 0,C 180,E1 -18056.014,E2 -18056.014} C_VEL
LIN {X 0,Y 286.349,Z 414.586,A -85,B 0,C 180,E1 -18058.151,E2 -18058.151} C_VEL
LIN {X 0,Y 280.385,Z 425.69,A -85,B 0,C 180,E1 -18060.74,E2 -18060.74} C_VEL
LIN {X 0,Y 275.769,Z 434.231,A -85,B 0,C 180,E1 -18063.178,E2 -18063.178} C_VEL
LIN {X 0,Y 270.97,Z 443.111,A -85,B 0,C 180,E1 -18066.296,E2 -18066.296} C_VEL
LIN {X 0,Y 267.495,Z 449.703,A -85,B 0,C 180,E1 -18069.225,E2 -18069.225} C_VEL
LIN {X 0,Y 264.812,Z 455.032,A -85,B 0,C 180,E1 -18072.229,E2 -18072.229} C_VEL
LIN {X 0,Y 263.773,Z 457.559,A -85,B 0,C 180,E1 -18073.776,E2 -18073.776} C_VEL
LIN {X 0,Y 262.409,Z 463.024,A -85,B 0,C 180,E1 -18076.841,E2 -18076.841} C_VEL
LIN {X 0,Y 261.679,Z 466.272,A -85,B 0,C 180,E1 -18079.164,E2 -18079.164} C_VEL
LIN {X 0,Y 261.205,Z 469.503,A -85,B 0,C 180,E1 -18082.269,E2 -18082.269} C_VEL
LIN {X 0,Y 261.065,Z 471.501,A -85,B 0,C 180,E1 -18085.368,E2 -18085.368} C_VEL
LIN {X 0,Y 261.127,Z 472.286,A -85,B 0,C 180,E1 -18088.458,E2 -18088.458} C_VEL
LIN {X 0,Y 261.131,Z 471.881,A -85,B 0,C 180,E1 -18091.542,E2 -18091.542} C_VEL
LIN {X 0,Y 261.065,Z 470.268,A -85,B 0,C 180,E1 -18094.632,E2 -18094.632} C_VEL
LIN {X 0,Y 261.204,Z 467.409,A -85,B 0,C 180,E1 -18097.731,E2 -18097.731} C_VEL
LIN {X 0,Y 261.57,Z 463.228,A -85,B 0,C 180,E1 -18100.841,E2 -18100.841} C_VEL
LIN {X 0,Y 262.248,Z 459.422,A -85,B 0,C 180,E1 -18103.167,E2 -18103.167} C_VEL
LIN {X 0,Y 263.73,Z 455.611,A -85,B 0,C 180,E1 -18106.395,E2 -18106.395} C_VEL
LIN {X 0,Y 265.96,Z 451.051,A -85,B 0,C 180,E1 -18109.288,E2 -18109.288} C_VEL
LIN {X 0,Y 269.038,Z 445.04,A -85,B 0,C 180,E1 -18112.258,E2 -18112.258} C_VEL
LIN {X 0,Y 272.851,Z 437.708,A -85,B 0,C 180,E1 -18115.151,E2 -18115.151} C_VEL
LIN {X 0,Y 277.549,Z 428.965,A -85,B 0,C 180,E1 -18117.934,E2 -18117.934} C_VEL
LIN {X 0,Y 283.211,Z 418.565,A -85,B 0,C 180,E1 -18120.578,E2 -18120.578} C_VEL
LIN {X 0,Y 289.664,Z 406.295,A -85,B 0,C 180,E1 -18123.087,E2 -18123.087} C_VEL
LIN {X 0,Y 296.01,Z 393.736,A -85,B 0,C 180,E1 -18125.153,E2 -18125.153} C_VEL
LIN {X 0,Y 303.55,Z 377.922,A -85,B 0,C 180,E1 -18127.219,E2 -18127.219} C_VEL
LIN {X 0,Y 309.658,Z 364.088,A -85,B 0,C 180,E1 -18128.619,E2 -18128.619} C_VEL
LIN {X 0,Y 315.617,Z 349.403,A -85,B 0,C 180,E1 -18129.806,E2 -18129.806} C_VEL
LIN {X 0,Y 321.949,Z 331.553,A -85,B 0,C 180,E1 -18130.911,E2 -18130.911} C_VEL
LIN {X 0,Y 327.2,Z 313.823,A -85,B 0,C 180,E1 -18131.748,E2 -18131.748} C_VEL
LIN {X 0,Y 346.201,Z 236.275,A -85,B 0,C 180,E1 -18134.775,E2 -18134.775} C_VEL
LIN {X 0,Y 346.192,Z 236.117,A -85,B 0,C 180,E1 -18136.022,E2 -18136.022} C_VEL
LIN {X 0,Y 331.1,Z 296.802,A -85,B 0,C 180,E1 -18138.358,E2 -18138.358} C_VEL
LIN {X 0,Y 326.673,Z 314.191,A -85,B 0,C 180,E1 -18139.196,E2 -18139.196} C_VEL
LIN {X 0,Y 322.065,Z 328.988,A -85,B 0,C 180,E1 -18140.133,E2 -18140.133} C_VEL
LIN {X 0,Y 316.542,Z 344.1,A -85,B 0,C 180,E1 -18141.359,E2 -18141.359} C_VEL
LIN {X 0,Y 310.811,Z 358.061,A -85,B 0,C 180,E1 -18142.781,E2 -18142.781} C_VEL
LIN {X 0,Y 304.056,Z 372.911,A -85,B 0,C 180,E1 -18144.701,E2 -18144.701} C_VEL
LIN {X 0,Y 297.77,Z 385.414,A -85,B 0,C 180,E1 -18146.719,E2 -18146.719} C_VEL
LIN {X 0,Y 291.129,Z 397.471,A -85,B 0,C 180,E1 -18149.138,E2 -18149.138} C_VEL
LIN {X 0,Y 285.23,Z 407.537,A -85,B 0,C 180,E1 -18151.686,E2 -18151.686} C_VEL
LIN {X 0,Y 280.612,Z 414.948,A -85,B 0,C 180,E1 -18154.006,E2 -18154.006} C_VEL
LIN {X 0,Y 275.736,Z 422.484,A -85,B 0,C 180,E1 -18156.977,E2 -18156.977} C_VEL
LIN {X 0,Y 272.068,Z 427.714,A -85,B 0,C 180,E1 -18159.591,E2 -18159.591} C_VEL
LIN {X 0,Y 269.485,Z 431.182,A -85,B 0,C 180,E1 -18161.763,E2 -18161.763} C_VEL
LIN {X 0,Y 266.733,Z 434.67,A -85,B 0,C 180,E1 -18164.724,E2 -18164.724} C_VEL
LIN {X 0,Y 264.766,Z 436.972,A -85,B 0,C 180,E1 -18167.74,E2 -18167.74} C_VEL
LIN {X 0,Y 263.172,Z 438.162,A -85,B 0,C 180,E1 -18170.78,E2 -18170.78} C_VEL
LIN {X 0,Y 262.129,Z 438.197,A -85,B 0,C 180,E1 -18173.844,E2 -18173.844} C_VEL
LIN {X 0,Y 261.628,Z 437.045,A -85,B 0,C 180,E1 -18176.921,E2 -18176.921} C_VEL
LIN {X 0,Y 261.321,Z 434.661,A -85,B 0,C 180,E1 -18180,E2 -18180} C_VEL
LIN {X 0,Y 261.332,Z 430.992,A -85,B 0,C 180,E1 -18183.084,E2 -18183.084} C_VEL
LIN {X 0,Y 261.472,Z 425.939,A -85,B 0,C 180,E1 -18186.173,E2 -18186.173} C_VEL
LIN {X 0,Y 261.912,Z 419.377,A -85,B 0,C 180,E1 -18189.265,E2 -18189.265} C_VEL
LIN {X 0,Y 262.461,Z 412.189,A -85,B 0,C 180,E1 -18191.978,E2 -18191.978} C_VEL
LIN {X 0,Y 263.318,Z 404.834,A -85,B 0,C 180,E1 -18194.294,E2 -18194.294} C_VEL
LIN {X 0,Y 264.416,Z 394.63,A -85,B 0,C 180,E1 -18197.001,E2 -18197.001} C_VEL
LIN {X 0,Y 265.732,Z 384.227,A -85,B 0,C 180,E1 -18199.306,E2 -18199.306} C_VEL
LIN {X 0,Y 267.451,Z 371.956,A -85,B 0,C 180,E1 -18201.586,E2 -18201.586} C_VEL
LIN {X 0,Y 269.032,Z 358.826,A -85,B 0,C 180,E1 -18203.621,E2 -18203.621} C_VEL
LIN {X 0,Y 270.745,Z 345.246,A -85,B 0,C 180,E1 -18205.361,E2 -18205.361} C_VEL
LIN {X 0,Y 272.466,Z 330.118,A -85,B 0,C 180,E1 -18206.937,E2 -18206.937} C_VEL
LIN {X 0,Y 273.961,Z 314.542,A -85,B 0,C 180,E1 -18208.229,E2 -18208.229} C_VEL
LIN {X 0,Y 275.258,Z 297.409,A -85,B 0,C 180,E1 -18209.312,E2 -18209.312} C_VEL
LIN {X 0,Y 276.441,Z 278.016,A -85,B 0,C 180,E1 -18210.169,E2 -18210.169} C_VEL
LIN {X 0,Y 282.178,Z 183.712,A -85,B 0,C 180,E1 -18213.779,E2 -18213.779} C_VEL
LIN {X 0,Y 265.231,Z 143.654,A -85,B 0,C 180,E1 -18216.992,E2 -18216.992} C_VEL
LIN {X 0,Y 263.229,Z 138.649,A -85,B 0,C 180,E1 -18217.415,E2 -18217.415} C_VEL
LIN {X 0,Y 263.182,Z 138.329,A -85,B 0,C 180,E1 -18217.504,E2 -18217.504} C_VEL
LIN {X 0,Y 263.11,Z 138.337,A -85,B 0,C 180,E1 -18221.897,E2 -18221.897} C_VEL
LIN {X 0,Y 263.08,Z 138.301,A -85,B 0,C 180,E1 -18226.162,E2 -18226.162} C_VEL
LIN {X 0,Y 263.115,Z 138.337,A -85,B 0,C 180,E1 -18230.771,E2 -18230.771} C_VEL
LIN {X 0,Y 263.159,Z 138.299,A -85,B 0,C 180,E1 -18234.017,E2 -18234.017} C_VEL
LIN {X 0,Y 263.131,Z 138.334,A -85,B 0,C 180,E1 -18237.711,E2 -18237.711} C_VEL
LIN {X 0,Y 263.149,Z 138.316,A -85,B 0,C 180,E1 -18241.806,E2 -18241.806} C_VEL
LIN {X 0,Y 263.117,Z 138.318,A -85,B 0,C 180,E1 -18246.381,E2 -18246.381} C_VEL
LIN {X 0,Y 263.21,Z 138.311,A -85,B 0,C 180,E1 -18249.689,E2 -18249.689} C_VEL
LIN {X 0,Y 263.186,Z 138.505,A -85,B 0,C 180,E1 -18251.421,E2 -18251.421} C_VEL
LIN {X 0,Y 266.208,Z 146.366,A -85,B 0,C 180,E1 -18253.667,E2 -18253.667} C_VEL
LIN {X 0,Y 273.627,Z 159.013,A -85,B 0,C 180,E1 -18255.353,E2 -18255.353} C_VEL
LIN {X 0,Y 283.262,Z 177.324,A -85,B 0,C 180,E1 -18257.434,E2 -18257.434} C_VEL
LIN {X 0,Y 292.699,Z 198.407,A -85,B 0,C 180,E1 -18259.41,E2 -18259.41} C_VEL
LIN {X 0,Y 293.071,Z 199.32,A -85,B 0,C 180,E1 -18259.486,E2 -18259.486} C_VEL
LIN {X 0,Y 288.014,Z 313.616,A -85,B 0,C 180,E1 -18262.331,E2 -18262.331} C_VEL
LIN {X 0,Y 286.679,Z 329.167,A -85,B 0,C 180,E1 -18262.959,E2 -18262.959} C_VEL
LIN {X 0,Y 284.968,Z 344.678,A -85,B 0,C 180,E1 -18263.895,E2 -18263.895} C_VEL
LIN {X 0,Y 282.805,Z 359.042,A -85,B 0,C 180,E1 -18265.037,E2 -18265.037} C_VEL
LIN {X 0,Y 280.483,Z 372.468,A -85,B 0,C 180,E1 -18266.409,E2 -18266.409} C_VEL
LIN {X 0,Y 277.824,Z 385.195,A -85,B 0,C 180,E1 -18268.007,E2 -18268.007} C_VEL
LIN {X 0,Y 274.955,Z 398.006,A -85,B 0,C 180,E1 -18270,E2 -18270} C_VEL
LIN {X 0,Y 272.165,Z 409.625,A -85,B 0,C 180,E1 -18272.22,E2 -18272.22} C_VEL
LIN {X 0,Y 269.632,Z 419.414,A -85,B 0,C 180,E1 -18274.485,E2 -18274.485} C_VEL
LIN {X 0,Y 267.131,Z 428.97,A -85,B 0,C 180,E1 -18277.179,E2 -18277.179} C_VEL
LIN {X 0,Y 265.139,Z 436.868,A -85,B 0,C 180,E1 -18279.921,E2 -18279.921} C_VEL
LIN {X 0,Y 263.371,Z 444.198,A -85,B 0,C 180,E1 -18283.11,E2 -18283.11} C_VEL
LIN {X 0,Y 262.184,Z 449.914,A -85,B 0,C 180,E1 -18286.347,E2 -18286.347} C_VEL
LIN {X 0,Y 261.498,Z 453.233,A -85,B 0,C 180,E1 -18288.815,E2 -18288.815} C_VEL
LIN {X 0,Y 260.924,Z 456.444,A -85,B 0,C 180,E1 -18292.154,E2 -18292.154} C_VEL
LIN {X 0,Y 260.761,Z 457.531,A -85,B 0,C 180,E1 -18293.846,E2 -18293.846} C_VEL
LIN {X 0,Y 260.663,Z 458.662,A -85,B 0,C 180,E1 -18297.281,E2 -18297.281} C_VEL
LIN {X 0,Y 260.823,Z 458.457,A -85,B 0,C 180,E1 -18300.428,E2 -18300.428} C_VEL
LIN {X 0,Y 261.213,Z 457.136,A -85,B 0,C 180,E1 -18303.481,E2 -18303.481} C_VEL
LIN {X 0,Y 261.941,Z 454.805,A -85,B 0,C 180,E1 -18306.397,E2 -18306.397} C_VEL
LIN {X 0,Y 263.231,Z 450.622,A -85,B 0,C 180,E1 -18309.85,E2 -18309.85} C_VEL
LIN {X 0,Y 264.676,Z 446,A -85,B 0,C 180,E1 -18312.636,E2 -18312.636} C_VEL
LIN {X 0,Y 266.554,Z 440.219,A -85,B 0,C 180,E1 -18315.389,E2 -18315.389} C_VEL
LIN {X 0,Y 268.984,Z 433.062,A -85,B 0,C 180,E1 -18318.129,E2 -18318.129} C_VEL
LIN {X 0,Y 272.013,Z 424.373,A -85,B 0,C 180,E1 -18320.815,E2 -18320.815} C_VEL
LIN {X 0,Y 274.883,Z 415.674,A -85,B 0,C 180,E1 -18323.033,E2 -18323.033} C_VEL
LIN {X 0,Y 278.117,Z 405.357,A -85,B 0,C 180,E1 -18325.213,E2 -18325.213} C_VEL
LIN {X 0,Y 281.584,Z 393.587,A -85,B 0,C 180,E1 -18327.243,E2 -18327.243} C_VEL
LIN {X 0,Y 284.915,Z 381.055,A -85,B 0,C 180,E1 -18329,E2 -18329} C_VEL
LIN {X 0,Y 288.099,Z 367.487,A -85,B 0,C 180,E1 -18330.526,E2 -18330.526} C_VEL
LIN {X 0,Y 289.069,Z 362.724,A -85,B 0,C 180,E1 -18330.994,E2 -18330.994} C_VEL
LIN {X 0,Y 288.789,Z 360.775,A -85,B 0,C 180,E1 -18331.278,E2 -18331.278} C_VEL
LIN {X 0,Y 287.101,Z 359.091,A -85,B 0,C 180,E1 -18331.763,E2 -18331.763} C_VEL
LIN {X 0,Y 283.827,Z 358.237,A -85,B 0,C 180,E1 -18332.425,E2 -18332.425} C_VEL
LIN {X 0,Y 280.854,Z 358.386,A -85,B 0,C 180,E1 -18332.926,E2 -18332.926} C_VEL
LIN {X 0,Y 265.37,Z 362.227,A -85,B 0,C 180,E1 -18335.372,E2 -18335.372} C_VEL
LIN {X 0,Y 263.839,Z 362.501,A -85,B 0,C 180,E1 -18335.654,E2 -18335.654} C_VEL
LIN {X 0,Y 262.002,Z 360.603,A -85,B 0,C 180,E1 -18336.378,E2 -18336.378} C_VEL
LIN {X 0,Y 260.356,Z 373.315,A -85,B 0,C 180,E1 -18338.42,E2 -18338.42} C_VEL
LIN {X 0,Y 258.811,Z 384.587,A -85,B 0,C 180,E1 -18340.57,E2 -18340.57} C_VEL
LIN {X 0,Y 257.295,Z 395.825,A -85,B 0,C 180,E1 -18343.125,E2 -18343.125} C_VEL
LIN {X 0,Y 256.291,Z 405.312,A -85,B 0,C 180,E1 -18345.711,E2 -18345.711} C_VEL
LIN {X 0,Y 255.286,Z 413.817,A -85,B 0,C 180,E1 -18348.486,E2 -18348.486} C_VEL
LIN {X 0,Y 254.728,Z 420.877,A -85,B 0,C 180,E1 -18351.271,E2 -18351.271} C_VEL
LIN {X 0,Y 254.378,Z 426.626,A -85,B 0,C 180,E1 -18354.052,E2 -18354.052} C_VEL
LIN {X 0,Y 254.289,Z 431.202,A -85,B 0,C 180,E1 -18356.831,E2 -18356.831} C_VEL
LIN {X 0,Y 254.249,Z 435.096,A -85,B 0,C 180,E1 -18359.999,E2 -18359.999} C_VEL
LIN {X 0,Y 254.587,Z 437.718,A -85,B 0,C 180,E1 -18363.164,E2 -18363.164} C_VEL
LIN {X 0,Y 255.124,Z 439.148,A -85,B 0,C 180,E1 -18366.326,E2 -18366.326} C_VEL
LIN {X 0,Y 256.284,Z 439.412,A -85,B 0,C 180,E1 -18369.47,E2 -18369.47} C_VEL
LIN {X 0,Y 257.875,Z 438.557,A -85,B 0,C 180,E1 -18372.593,E2 -18372.593} C_VEL
LIN {X 0,Y 259.966,Z 436.547,A -85,B 0,C 180,E1 -18375.684,E2 -18375.684} C_VEL
LIN {X 0,Y 262.918,Z 433.361,A -85,B 0,C 180,E1 -18378.709,E2 -18378.709} C_VEL
LIN {X 0,Y 266.542,Z 429.009,A -85,B 0,C 180,E1 -18381.662,E2 -18381.662} C_VEL
LIN {X 0,Y 270.903,Z 423.421,A -85,B 0,C 180,E1 -18384.524,E2 -18384.524} C_VEL
LIN {X 0,Y 275.931,Z 416.512,A -85,B 0,C 180,E1 -18387.288,E2 -18387.288} C_VEL
LIN {X 0,Y 281.673,Z 408.119,A -85,B 0,C 180,E1 -18389.935,E2 -18389.935} C_VEL
LIN {X 0,Y 288.119,Z 398.096,A -85,B 0,C 180,E1 -18392.455,E2 -18392.455} C_VEL
LIN {X 0,Y 295.131,Z 386.249,A -85,B 0,C 180,E1 -18394.856,E2 -18394.856} C_VEL
LIN {X 0,Y 301.963,Z 373.92,A -85,B 0,C 180,E1 -18396.821,E2 -18396.821} C_VEL
LIN {X 0,Y 308.316,Z 361.246,A -85,B 0,C 180,E1 -18398.469,E2 -18398.469} C_VEL
LIN {X 0,Y 314.294,Z 348.173,A -85,B 0,C 180,E1 -18399.85,E2 -18399.85} C_VEL
LIN {X 0,Y 320.555,Z 332.703,A -85,B 0,C 180,E1 -18401.127,E2 -18401.127} C_VEL
LIN {X 0,Y 325.386,Z 318.919,A -85,B 0,C 180,E1 -18402.033,E2 -18402.033} C_VEL
LIN {X 0,Y 330.278,Z 302.215,A -85,B 0,C 180,E1 -18402.876,E2 -18402.876} C_VEL
LIN {X 0,Y 341.099,Z 260.972,A -85,B 0,C 180,E1 -18404.47,E2 -18404.47} C_VEL
LIN {X 0,Y 341.114,Z 260.95,A -85,B 0,C 180,E1 -18404.679,E2 -18404.679} C_VEL
LIN {X 0,Y 327.464,Z 313.584,A -85,B 0,C 180,E1 -18406.73,E2 -18406.73} C_VEL
LIN {X 0,Y 321.645,Z 331.721,A -85,B 0,C 180,E1 -18407.575,E2 -18407.575} C_VEL
LIN {X 0,Y 315.678,Z 347.446,A -85,B 0,C 180,E1 -18408.522,E2 -18408.522} C_VEL
LIN {X 0,Y 309.334,Z 362.192,A -85,B 0,C 180,E1 -18409.646,E2 -18409.646} C_VEL
LIN {X 0,Y 302.229,Z 377.116,A -85,B 0,C 180,E1 -18411.108,E2 -18411.108} C_VEL
LIN {X 0,Y 295.73,Z 389.869,A -85,B 0,C 180,E1 -18412.699,E2 -18412.699} C_VEL
LIN {X 0,Y 288.668,Z 402.812,A -85,B 0,C 180,E1 -18414.674,E2 -18414.674} C_VEL
LIN {X 0,Y 282.319,Z 413.991,A -85,B 0,C 180,E1 -18416.793,E2 -18416.793} C_VEL
LIN {X 0,Y 275.909,Z 424.96,A -85,B 0,C 180,E1 -18419.373,E2 -18419.373} C_VEL
LIN {X 0,Y 270.282,Z 434.339,A -85,B 0,C 180,E1 -18422.093,E2 -18422.093} C_VEL
LIN {X 0,Y 265.551,Z 442.265,A -85,B 0,C 180,E1 -18424.947,E2 -18424.947} C_VEL
LIN {X 0,Y 261.72,Z 448.836,A -85,B 0,C 180,E1 -18427.917,E2 -18427.917} C_VEL
LIN {X 0,Y 258.637,Z 454.187,A -85,B 0,C 180,E1 -18430.969,E2 -18430.969} C_VEL
LIN {X 0,Y 256.954,Z 457.3,A -85,B 0,C 180,E1 -18433.193,E2 -18433.193} C_VEL
LIN {X 0,Y 255.433,Z 462.992,A -85,B 0,C 180,E1 -18436.475,E2 -18436.475} C_VEL
LIN {X 0,Y 254.635,Z 466.196,A -85,B 0,C 180,E1 -18438.86,E2 -18438.86} C_VEL
LIN {X 0,Y 254.129,Z 469.385,A -85,B 0,C 180,E1 -18442.052,E2 -18442.052} C_VEL
LIN {X 0,Y 253.972,Z 471.358,A -85,B 0,C 180,E1 -18445.238,E2 -18445.238} C_VEL
LIN {X 0,Y 254.032,Z 472.109,A -85,B 0,C 180,E1 -18448.415,E2 -18448.415} C_VEL
LIN {X 0,Y 254.037,Z 471.668,A -85,B 0,C 180,E1 -18451.585,E2 -18451.585} C_VEL
LIN {X 0,Y 253.972,Z 470.019,A -85,B 0,C 180,E1 -18454.762,E2 -18454.762} C_VEL
LIN {X 0,Y 254.126,Z 467.121,A -85,B 0,C 180,E1 -18457.948,E2 -18457.948} C_VEL
LIN {X 0,Y 254.526,Z 462.898,A -85,B 0,C 180,E1 -18461.145,E2 -18461.145} C_VEL
LIN {X 0,Y 255.117,Z 459.724,A -85,B 0,C 180,E1 -18463.137,E2 -18463.137} C_VEL
LIN {X 0,Y 256.797,Z 456.051,A -85,B 0,C 180,E1 -18466.69,E2 -18466.69} C_VEL
LIN {X 0,Y 259.259,Z 451.545,A -85,B 0,C 180,E1 -18469.807,E2 -18469.807} C_VEL
LIN {X 0,Y 262.515,Z 445.817,A -85,B 0,C 180,E1 -18472.842,E2 -18472.842} C_VEL
LIN {X 0,Y 266.539,Z 438.852,A -85,B 0,C 180,E1 -18475.789,E2 -18475.789} C_VEL
LIN {X 0,Y 271.448,Z 430.523,A -85,B 0,C 180,E1 -18478.619,E2 -18478.619} C_VEL
LIN {X 0,Y 278.16,Z 419.306,A -85,B 0,C 180,E1 -18481.619,E2 -18481.619} C_VEL
LIN {X 0,Y 284.962,Z 407.476,A -85,B 0,C 180,E1 -18484.131,E2 -18484.131} C_VEL
LIN {X 0,Y 291.619,Z 395.369,A -85,B 0,C 180,E1 -18486.189,E2 -18486.189} C_VEL
LIN {X 0,Y 298.393,Z 382.363,A -85,B 0,C 180,E1 -18487.975,E2 -18487.975} C_VEL
LIN {X 0,Y 304.638,Z 369.68,A -85,B 0,C 180,E1 -18489.377,E2 -18489.377} C_VEL
LIN {X 0,Y 311.344,Z 354.768,A -85,B 0,C 180,E1 -18490.677,E2 -18490.677} C_VEL
LIN {X 0,Y 317.123,Z 340.349,A -85,B 0,C 180,E1 -18491.671,E2 -18491.671} C_VEL
LIN {X 0,Y 322.888,Z 324.055,A -85,B 0,C 180,E1 -18492.54,E2 -18492.54} C_VEL
LIN {X 0,Y 328.828,Z 303.192,A -85,B 0,C 180,E1 -18493.441,E2 -18493.441} C_VEL
LIN {X 0,Y 341.735,Z 252.712,A -85,B 0,C 180,E1 -18495.382,E2 -18495.382} C_VEL
LIN {X 0,Y 341.707,Z 252.791,A -85,B 0,C 180,E1 -18495.441,E2 -18495.441} C_VEL
LIN {X 0,Y 327.94,Z 305.911,A -85,B 0,C 180,E1 -18497.512,E2 -18497.512} C_VEL
LIN {X 0,Y 323.509,Z 320.675,A -85,B 0,C 180,E1 -18498.295,E2 -18498.295} C_VEL
LIN {X 0,Y 318.179,Z 335.812,A -85,B 0,C 180,E1 -18499.338,E2 -18499.338} C_VEL
LIN {X 0,Y 312.221,Z 350.356,A -85,B 0,C 180,E1 -18500.618,E2 -18500.618} C_VEL
LIN {X 0,Y 306.528,Z 362.695,A -85,B 0,C 180,E1 -18501.962,E2 -18501.962} C_VEL
LIN {X 0,Y 299.976,Z 375.727,A -85,B 0,C 180,E1 -18503.732,E2 -18503.732} C_VEL
LIN {X 0,Y 293.381,Z 387.735,A -85,B 0,C 180,E1 -18505.741,E2 -18505.741} C_VEL
LIN {X 0,Y 286.407,Z 399.406,A -85,B 0,C 180,E1 -18508.158,E2 -18508.158} C_VEL
LIN {X 0,Y 280.163,Z 409.176,A -85,B 0,C 180,E1 -18510.715,E2 -18510.715} C_VEL
LIN {X 0,Y 274.605,Z 417.306,A -85,B 0,C 180,E1 -18513.393,E2 -18513.393} C_VEL
LIN {X 0,Y 269.826,Z 423.943,A -85,B 0,C 180,E1 -18516.19,E2 -18516.19} C_VEL
LIN {X 0,Y 265.599,Z 429.33,A -85,B 0,C 180,E1 -18519.071,E2 -18519.071} C_VEL
LIN {X 0,Y 262.877,Z 432.549,A -85,B 0,C 180,E1 -18521.288,E2 -18521.288} C_VEL
LIN {X 0,Y 259.97,Z 435.801,A -85,B 0,C 180,E1 -18524.316,E2 -18524.316} C_VEL
LIN {X 0,Y 257.87,Z 437.851,A -85,B 0,C 180,E1 -18527.407,E2 -18527.407} C_VEL
LIN {X 0,Y 256.181,Z 438.788,A -85,B 0,C 180,E1 -18530.526,E2 -18530.526} C_VEL
LIN {X 0,Y 255.084,Z 438.58,A -85,B 0,C 180,E1 -18533.673,E2 -18533.673} C_VEL
LIN {X 0,Y 254.557,Z 437.205,A -85,B 0,C 180,E1 -18536.835,E2 -18536.835} C_VEL
LIN {X 0,Y 254.241,Z 434.628,A -85,B 0,C 180,E1 -18540.001,E2 -18540.001} C_VEL
LIN {X 0,Y 254.245,Z 430.765,A -85,B 0,C 180,E1 -18543.17,E2 -18543.17} C_VEL
LIN {X 0,Y 254.414,Z 425.487,A -85,B 0,C 180,E1 -18546.344,E2 -18546.344} C_VEL
LIN {X 0,Y 254.854,Z 418.657,A -85,B 0,C 180,E1 -18549.524,E2 -18549.524} C_VEL
LIN {X 0,Y 255.468,Z 411.237,A -85,B 0,C 180,E1 -18552.311,E2 -18552.311} C_VEL
LIN {X 0,Y 256.34,Z 403.671,A -85,B 0,C 180,E1 -18554.691,E2 -18554.691} C_VEL
LIN {X 0,Y 257.536,Z 393.159,A -85,B 0,C 180,E1 -18557.469,E2 -18557.469} C_VEL
LIN {X 0,Y 259.068,Z 381.409,A -85,B 0,C 180,E1 -18560.029,E2 -18560.029} C_VEL
LIN {X 0,Y 260.816,Z 368.436,A -85,B 0,C 180,E1 -18562.372,E2 -18562.372} C_VEL
LIN {X 0,Y 262.533,Z 355.407,A -85,B 0,C 180,E1 -18564.331,E2 -18564.331} C_VEL
LIN {X 0,Y 264.18,Z 341.745,A -85,B 0,C 180,E1 -18566.038,E2 -18566.038} C_VEL
LIN {X 0,Y 265.84,Z 326.811,A -85,B 0,C 180,E1 -18567.559,E2 -18567.559} C_VEL
LIN {X 0,Y 267.29,Z 311.702,A -85,B 0,C 180,E1 -18568.784,E2 -18568.784} C_VEL
LIN {X 0,Y 268.539,Z 294.956,A -85,B 0,C 180,E1 -18569.819,E2 -18569.819} C_VEL
LIN {X 0,Y 270.852,Z 257.627,A -85,B 0,C 180,E1 -18571.372,E2 -18571.372} C_VEL
LIN {X 0,Y 275.512,Z 185.621,A -85,B 0,C 180,E1 -18574.218,E2 -18574.218} C_VEL
LIN {X 0,Y 259.37,Z 147.292,A -85,B 0,C 180,E1 -18577.36,E2 -18577.36} C_VEL
LIN {X 0,Y 256.149,Z 139.407,A -85,B 0,C 180,E1 -18578.047,E2 -18578.047} C_VEL
LIN {X 0,Y 256.057,Z 139.214,A -85,B 0,C 180,E1 -18582.177,E2 -18582.177} C_VEL
LIN {X 0,Y 256.024,Z 139.178,A -85,B 0,C 180,E1 -18586.665,E2 -18586.665} C_VEL
LIN {X 0,Y 256.069,Z 139.215,A -85,B 0,C 180,E1 -18590.857,E2 -18590.857} C_VEL
LIN {X 0,Y 256.128,Z 139.184,A -85,B 0,C 180,E1 -18592.867,E2 -18592.867} C_VEL
LIN {X 0,Y 256.069,Z 139.208,A -85,B 0,C 180,E1 -18596.707,E2 -18596.707} C_VEL
LIN {X 0,Y 256.057,Z 139.191,A -85,B 0,C 180,E1 -18600.393,E2 -18600.393} C_VEL
LIN {X 0,Y 256.081,Z 139.21,A -85,B 0,C 180,E1 -18603.953,E2 -18603.953} C_VEL
LIN {X 0,Y 256.059,Z 139.207,A -85,B 0,C 180,E1 -18607.402,E2 -18607.402} C_VEL
LIN {X 0,Y 256.137,Z 139.264,A -85,B 0,C 180,E1 -18610.203,E2 -18610.203} C_VEL
LIN {X 0,Y 258.921,Z 146.432,A -85,B 0,C 180,E1 -18612.364,E2 -18612.364} C_VEL
LIN {X 0,Y 267.2,Z 160.456,A -85,B 0,C 180,E1 -18614.343,E2 -18614.343} C_VEL
LIN {X 0,Y 276.836,Z 178.512,A -85,B 0,C 180,E1 -18616.518,E2 -18616.518} C_VEL
LIN {X 0,Y 283.253,Z 192.483,A -85,B 0,C 180,E1 -18617.924,E2 -18617.924} C_VEL
LIN {X 0,Y 287.15,Z 201.451,A -85,B 0,C 180,E1 -18618.757,E2 -18618.757} C_VEL
LIN {X 0,Y 281.963,Z 313.339,A -85,B 0,C 180,E1 -18621.58,E2 -18621.58} C_VEL
LIN {X 0,Y 280.609,Z 329.011,A -85,B 0,C 180,E1 -18622.218,E2 -18622.218} C_VEL
LIN {X 0,Y 278.896,Z 344.035,A -85,B 0,C 180,E1 -18623.125,E2 -18623.125} C_VEL
LIN {X 0,Y 276.705,Z 358.59,A -85,B 0,C 180,E1 -18624.294,E2 -18624.294} C_VEL
LIN {X 0,Y 274.388,Z 371.374,A -85,B 0,C 180,E1 -18625.593,E2 -18625.593} C_VEL
LIN {X 0,Y 271.676,Z 384.295,A -85,B 0,C 180,E1 -18627.22,E2 -18627.22} C_VEL
LIN {X 0,Y 268.924,Z 396.235,A -85,B 0,C 180,E1 -18629.064,E2 -18629.064} C_VEL
LIN {X 0,Y 266.112,Z 407.574,A -85,B 0,C 180,E1 -18631.196,E2 -18631.196} C_VEL
LIN {X 0,Y 263.506,Z 417.475,A -85,B 0,C 180,E1 -18633.44,E2 -18633.44} C_VEL
LIN {X 0,Y 261.308,Z 425.596,A -85,B 0,C 180,E1 -18635.649,E2 -18635.649} C_VEL
LIN {X 0,Y 258.906,Z 434.538,A -85,B 0,C 180,E1 -18638.586,E2 -18638.586} C_VEL
LIN {X 0,Y 257.33,Z 440.561,A -85,B 0,C 180,E1 -18641.022,E2 -18641.022} C_VEL
LIN {X 0,Y 255.786,Z 447.136,A -85,B 0,C 180,E1 -18644.317,E2 -18644.317} C_VEL
LIN {X 0,Y 254.72,Z 452.188,A -85,B 0,C 180,E1 -18647.668,E2 -18647.668} C_VEL
LIN {X 0,Y 253.949,Z 455.831,A -85,B 0,C 180,E1 -18651.086,E2 -18651.086} C_VEL
LIN {X 0,Y 253.62,Z 458.076,A -85,B 0,C 180,E1 -18654.561,E2 -18654.561} C_VEL
LIN {X 0,Y 253.576,Z 458.932,A -85,B 0,C 180,E1 -18658.11,E2 -18658.11} C_VEL
LIN {X 0,Y 253.751,Z 458.586,A -85,B 0,C 180,E1 -18660.84,E2 -18660.84} C_VEL
LIN {X 0,Y 254.235,Z 457.184,A -85,B 0,C 180,E1 -18663.971,E2 -18663.971} C_VEL
LIN {X 0,Y 255.122,Z 454.434,A -85,B 0,C 180,E1 -18667.304,E2 -18667.304} C_VEL
LIN {X 0,Y 256.1,Z 451.491,A -85,B 0,C 180,E1 -18669.79,E2 -18669.79} C_VEL
LIN {X 0,Y 257.755,Z 446.516,A -85,B 0,C 180,E1 -18672.973,E2 -18672.973} C_VEL
LIN {X 0,Y 259.81,Z 440.591,A -85,B 0,C 180,E1 -18675.904,E2 -18675.904} C_VEL
LIN {X 0,Y 262.287,Z 433.756,A -85,B 0,C 180,E1 -18678.613,E2 -18678.613} C_VEL
LIN {X 0,Y 265.449,Z 425.185,A -85,B 0,C 180,E1 -18681.356,E2 -18681.356} C_VEL
LIN {X 0,Y 268.558,Z 416.214,A -85,B 0,C 180,E1 -18683.713,E2 -18683.713} C_VEL
LIN {X 0,Y 272.161,Z 405.31,A -85,B 0,C 180,E1 -18686.054,E2 -18686.054} C_VEL
LIN {X 0,Y 275.959,Z 392.894,A -85,B 0,C 180,E1 -18688.21,E2 -18688.21} C_VEL
LIN {X 0,Y 279.286,Z 380.77,A -85,B 0,C 180,E1 -18689.921,E2 -18689.921} C_VEL
LIN {X 0,Y 282.494,Z 367.577,A -85,B 0,C 180,E1 -18691.421,E2 -18691.421} C_VEL
LIN {X 0,Y 284.341,Z 358.776,A -85,B 0,C 180,E1 -18692.258,E2 -18692.258} C_VEL
LIN {X 0,Y 281.063,Z 360.023,A -85,B 0,C 180,E1 -18692.667,E2 -18692.667} C_VEL
LIN {X 0,Y 265.37,Z 362.227,A -85,B 0,C 180,E1 -18695.372,E2 -18695.372} C_VEL
LIN {X 0,Y 262.558,Z 363.197,A -85,B 0,C 180,E1 -18695.919,E2 -18695.919} C_VEL
LIN {X 0,Y 258.953,Z 365.931,A -85,B 0,C 180,E1 -18696.743,E2 -18696.743} C_VEL
LIN {X 0,Y 256.136,Z 369.658,A -85,B 0,C 180,E1 -18697.555,E2 -18697.555} C_VEL
LIN {X 0,Y 253.469,Z 375.682,A -85,B 0,C 180,E1 -18698.666,E2 -18698.666} C_VEL
LIN {X 0,Y 252.105,Z 381.801,A -85,B 0,C 180,E1 -18699.841,E2 -18699.841} C_VEL
LIN {X 0,Y 250.534,Z 393.757,A -85,B 0,C 180,E1 -18702.511,E2 -18702.511} C_VEL
LIN {X 0,Y 249.332,Z 404.111,A -85,B 0,C 180,E1 -18705.304,E2 -18705.304} C_VEL
LIN {X 0,Y 248.28,Z 412.888,A -85,B 0,C 180,E1 -18708.157,E2 -18708.157} C_VEL
LIN {X 0,Y 247.677,Z 420.2,A -85,B 0,C 180,E1 -18711.021,E2 -18711.021} C_VEL
LIN {X 0,Y 247.284,Z 426.593,A -85,B 0,C 180,E1 -18714.114,E2 -18714.114} C_VEL
LIN {X 0,Y 247.199,Z 432.089,A -85,B 0,C 180,E1 -18717.555,E2 -18717.555} C_VEL
LIN {X 0,Y 247.171,Z 435.021,A -85,B 0,C 180,E1 -18719.999,E2 -18719.999} C_VEL
LIN {X 0,Y 247.518,Z 437.874,A -85,B 0,C 180,E1 -18723.255,E2 -18723.255} C_VEL
LIN {X 0,Y 248.085,Z 439.541,A -85,B 0,C 180,E1 -18726.506,E2 -18726.506} C_VEL
LIN {X 0,Y 249.304,Z 440.034,A -85,B 0,C 180,E1 -18729.737,E2 -18729.737} C_VEL
LIN {X 0,Y 250.999,Z 439.363,A -85,B 0,C 180,E1 -18732.944,E2 -18732.944} C_VEL
LIN {X 0,Y 253.219,Z 437.616,A -85,B 0,C 180,E1 -18736.113,E2 -18736.113} C_VEL
LIN {X 0,Y 256.35,Z 434.731,A -85,B 0,C 180,E1 -18739.207,E2 -18739.207} C_VEL
LIN {X 0,Y 260.154,Z 430.714,A -85,B 0,C 180,E1 -18742.222,E2 -18742.222} C_VEL
LIN {X 0,Y 265.47,Z 424.579,A -85,B 0,C 180,E1 -18745.549,E2 -18745.549} C_VEL
LIN {X 0,Y 271.426,Z 417.082,A -85,B 0,C 180,E1 -18748.621,E2 -18748.621} C_VEL
LIN {X 0,Y 277.615,Z 408.795,A -85,B 0,C 180,E1 -18751.263,E2 -18751.263} C_VEL
LIN {X 0,Y 284.498,Z 398.911,A -85,B 0,C 180,E1 -18753.767,E2 -18753.767} C_VEL
LIN {X 0,Y 291.973,Z 387.285,A -85,B 0,C 180,E1 -18756.138,E2 -18756.138} C_VEL
LIN {X 0,Y 299.172,Z 375.203,A -85,B 0,C 180,E1 -18758.072,E2 -18758.072} C_VEL
LIN {X 0,Y 306.237,Z 362.185,A -85,B 0,C 180,E1 -18759.77,E2 -18759.77} C_VEL
LIN {X 0,Y 313.175,Z 347.917,A -85,B 0,C 180,E1 -18761.239,E2 -18761.239} C_VEL
LIN {X 0,Y 319.95,Z 332.138,A -85,B 0,C 180,E1 -18762.489,E2 -18762.489} C_VEL
LIN {X 0,Y 325.035,Z 318.306,A -85,B 0,C 180,E1 -18763.354,E2 -18763.354} C_VEL
LIN {X 0,Y 329.772,Z 302.901,A -85,B 0,C 180,E1 -18764.103,E2 -18764.103} C_VEL
LIN {X 0,Y 332.781,Z 291.787,A -85,B 0,C 180,E1 -18764.541,E2 -18764.541} C_VEL
LIN {X 0,Y 332.829,Z 291.613,A -85,B 0,C 180,E1 -18764.612,E2 -18764.612} C_VEL
LIN {X 0,Y 327.204,Z 312.117,A -85,B 0,C 180,E1 -18765.405,E2 -18765.405} C_VEL
LIN {X 0,Y 321.465,Z 329.261,A -85,B 0,C 180,E1 -18766.175,E2 -18766.175} C_VEL
LIN {X 0,Y 314.927,Z 345.734,A -85,B 0,C 180,E1 -18767.106,E2 -18767.106} C_VEL
LIN {X 0,Y 307.627,Z 361.77,A -85,B 0,C 180,E1 -18768.288,E2 -18768.288} C_VEL
LIN {X 0,Y 299.542,Z 377.531,A -85,B 0,C 180,E1 -18769.818,E2 -18769.818} C_VEL
LIN {X 0,Y 292.678,Z 390.003,A -85,B 0,C 180,E1 -18771.367,E2 -18771.367} C_VEL
LIN {X 0,Y 284.25,Z 404.273,A -85,B 0,C 180,E1 -18773.602,E2 -18773.602} C_VEL
LIN {X 0,Y 276.675,Z 416.452,A -85,B 0,C 180,E1 -18776.025,E2 -18776.025} C_VEL
LIN {X 0,Y 269.24,Z 428.068,A -85,B 0,C 180,E1 -18778.967,E2 -18778.967} C_VEL
LIN {X 0,Y 263.564,Z 436.689,A -85,B 0,C 180,E1 -18781.726,E2 -18781.726} C_VEL
LIN {X 0,Y 259.193,Z 443.24,A -85,B 0,C 180,E1 -18784.289,E2 -18784.289} C_VEL
LIN {X 0,Y 255.173,Z 449.5,A -85,B 0,C 180,E1 -18787.32,E2 -18787.32} C_VEL
LIN {X 0,Y 251.923,Z 454.596,A -85,B 0,C 180,E1 -18790.441,E2 -18790.441} C_VEL
LIN {X 0,Y 249.98,Z 457.716,A -85,B 0,C 180,E1 -18792.916,E2 -18792.916} C_VEL
LIN {X 0,Y 248.473,Z 462.959,A -85,B 0,C 180,E1 -18796.089,E2 -18796.089} C_VEL
LIN {X 0,Y 247.603,Z 466.12,A -85,B 0,C 180,E1 -18798.54,E2 -18798.54} C_VEL
LIN {X 0,Y 247.072,Z 469.268,A -85,B 0,C 180,E1 -18801.823,E2 -18801.823} C_VEL
LIN {X 0,Y 246.88,Z 471.21,A -85,B 0,C 180,E1 -18805.101,E2 -18805.101} C_VEL
LIN {X 0,Y 246.938,Z 471.932,A -85,B 0,C 180,E1 -18808.369,E2 -18808.369} C_VEL
LIN {X 0,Y 246.987,Z 471.842,A -85,B 0,C 180,E1 -18810,E2 -18810} C_VEL
LIN {X 0,Y 246.9,Z 470.759,A -85,B 0,C 180,E1 -18813.264,E2 -18813.264} C_VEL
LIN {X 0,Y 246.955,Z 468.451,A -85,B 0,C 180,E1 -18816.536,E2 -18816.536} C_VEL
LIN {X 0,Y 247.243,Z 464.855,A -85,B 0,C 180,E1 -18819.82,E2 -18819.82} C_VEL
LIN {X 0,Y 247.988,Z 459.923,A -85,B 0,C 180,E1 -18823.104,E2 -18823.104} C_VEL
LIN {X 0,Y 249.804,Z 456.458,A -85,B 0,C 180,E1 -18826.952,E2 -18826.952} C_VEL
LIN {X 0,Y 252.576,Z 451.991,A -85,B 0,C 180,E1 -18830.354,E2 -18830.354} C_VEL
LIN {X 0,Y 256.029,Z 446.602,A -85,B 0,C 180,E1 -18833.455,E2 -18833.455} C_VEL
LIN {X 0,Y 260.254,Z 440.004,A -85,B 0,C 180,E1 -18836.46,E2 -18836.46} C_VEL
LIN {X 0,Y 265.412,Z 432.099,A -85,B 0,C 180,E1 -18839.332,E2 -18839.332} C_VEL
LIN {X 0,Y 271.558,Z 422.751,A -85,B 0,C 180,E1 -18842.042,E2 -18842.042} C_VEL
LIN {X 0,Y 278.513,Z 411.779,A -85,B 0,C 180,E1 -18844.595,E2 -18844.595} C_VEL
LIN {X 0,Y 285.313,Z 400.65,A -85,B 0,C 180,E1 -18846.68,E2 -18846.68} C_VEL
LIN {X 0,Y 293.305,Z 386.76,A -85,B 0,C 180,E1 -18848.755,E2 -18848.755} C_VEL
LIN {X 0,Y 300.228,Z 373.872,A -85,B 0,C 180,E1 -18850.291,E2 -18850.291} C_VEL
LIN {X 0,Y 307.75,Z 358.665,A -85,B 0,C 180,E1 -18851.692,E2 -18851.692} C_VEL
LIN {X 0,Y 314.445,Z 343.641,A -85,B 0,C 180,E1 -18852.758,E2 -18852.758} C_VEL
LIN {X 0,Y 320.727,Z 327.505,A -85,B 0,C 180,E1 -18853.649,E2 -18853.649} C_VEL
LIN {X 0,Y 326.544,Z 309.318,A -85,B 0,C 180,E1 -18854.448,E2 -18854.448} C_VEL
LIN {X 0,Y 333.082,Z 284.978,A -85,B 0,C 180,E1 -18855.398,E2 -18855.398} C_VEL
LIN {X 0,Y 326.449,Z 309.433,A -85,B 0,C 180,E1 -18856.403,E2 -18856.403} C_VEL
LIN {X 0,Y 321.138,Z 325.394,A -85,B 0,C 180,E1 -18857.28,E2 -18857.28} C_VEL
LIN {X 0,Y 315.585,Z 339.561,A -85,B 0,C 180,E1 -18858.294,E2 -18858.294} C_VEL
LIN {X 0,Y 309.088,Z 354.011,A -85,B 0,C 180,E1 -18859.607,E2 -18859.607} C_VEL
LIN {X 0,Y 302.362,Z 367.329,A -85,B 0,C 180,E1 -18861.129,E2 -18861.129} C_VEL
LIN {X 0,Y 295.031,Z 380.524,A -85,B 0,C 180,E1 -18863.024,E2 -18863.024} C_VEL
LIN {X 0,Y 288.189,Z 391.761,A -85,B 0,C 180,E1 -18865.034,E2 -18865.034} C_VEL
LIN {X 0,Y 280.905,Z 402.719,A -85,B 0,C 180,E1 -18867.459,E2 -18867.459} C_VEL
LIN {X 0,Y 275.181,Z 410.872,A -85,B 0,C 180,E1 -18869.709,E2 -18869.709} C_VEL
LIN {X 0,Y 269.966,Z 417.85,A -85,B 0,C 180,E1 -18872.057,E2 -18872.057} C_VEL
LIN {X 0,Y 264.795,Z 424.436,A -85,B 0,C 180,E1 -18874.871,E2 -18874.871} C_VEL
LIN {X 0,Y 260.184,Z 429.767,A -85,B 0,C 180,E1 -18877.781,E2 -18877.781} C_VEL
LIN {X 0,Y 256.286,Z 433.901,A -85,B 0,C 180,E1 -18880.788,E2 -18880.788} C_VEL
LIN {X 0,Y 253.221,Z 436.852,A -85,B 0,C 180,E1 -18883.887,E2 -18883.887} C_VEL
LIN {X 0,Y 250.989,Z 438.674,A -85,B 0,C 180,E1 -18887.056,E2 -18887.056} C_VEL
LIN {X 0,Y 249.213,Z 439.409,A -85,B 0,C 180,E1 -18890.259,E2 -18890.259} C_VEL
LIN {X 0,Y 248.045,Z 438.959,A -85,B 0,C 180,E1 -18893.493,E2 -18893.493} C_VEL
LIN {X 0,Y 247.488,Z 437.348,A -85,B 0,C 180,E1 -18896.745,E2 -18896.745} C_VEL
LIN {X 0,Y 247.162,Z 434.542,A -85,B 0,C 180,E1 -18900.001,E2 -18900.001} C_VEL
LIN {X 0,Y 247.159,Z 430.447,A -85,B 0,C 180,E1 -18903.261,E2 -18903.261} C_VEL
LIN {X 0,Y 247.343,Z 424.939,A -85,B 0,C 180,E1 -18906.527,E2 -18906.527} C_VEL
LIN {X 0,Y 247.672,Z 419.819,A -85,B 0,C 180,E1 -18908.979,E2 -18908.979} C_VEL
LIN {X 0,Y 248.345,Z 411.368,A -85,B 0,C 180,E1 -18912.254,E2 -18912.254} C_VEL
LIN {X 0,Y 249.365,Z 402.355,A -85,B 0,C 180,E1 -18915.112,E2 -18915.112} C_VEL
LIN {X 0,Y 250.5,Z 392.775,A -85,B 0,C 180,E1 -18917.652,E2 -18917.652} C_VEL
LIN {X 0,Y 252.002,Z 381.347,A -85,B 0,C 180,E1 -18920.19,E2 -18920.19} C_VEL
LIN {X 0,Y 253.789,Z 368.315,A -85,B 0,C 180,E1 -18922.597,E2 -18922.597} C_VEL
LIN {X 0,Y 255.543,Z 355.312,A -85,B 0,C 180,E1 -18924.594,E2 -18924.594} C_VEL
LIN {X 0,Y 257.252,Z 341.5,A -85,B 0,C 180,E1 -18926.356,E2 -18926.356} C_VEL
LIN {X 0,Y 258.955,Z 326.443,A -85,B 0,C 180,E1 -18927.916,E2 -18927.916} C_VEL
LIN {X 0,Y 260.445,Z 311.182,A -85,B 0,C 180,E1 -18929.171,E2 -18929.171} C_VEL
LIN {X 0,Y 261.745,Z 294.137,A -85,B 0,C 180,E1 -18930.229,E2 -18930.229} C_VEL
LIN {X 0,Y 267.567,Z 204.264,A -85,B 0,C 180,E1 -18933.989,E2 -18933.989} C_VEL
LIN {X 0,Y 268.724,Z 187.203,A -85,B 0,C 180,E1 -18934.678,E2 -18934.678} C_VEL
LIN {X 0,Y 253.03,Z 149.864,A -85,B 0,C 180,E1 -18937.827,E2 -18937.827} C_VEL
LIN {X 0,Y 249.159,Z 140.637,A -85,B 0,C 180,E1 -18938.67,E2 -18938.67} C_VEL
LIN {X 0,Y 249.051,Z 140.087,A -85,B 0,C 180,E1 -18938.772,E2 -18938.772} C_VEL
LIN {X 0,Y 248.986,Z 140.096,A -85,B 0,C 180,E1 -18942.786,E2 -18942.786} C_VEL
LIN {X 0,Y 248.981,Z 140.057,A -85,B 0,C 180,E1 -18947.355,E2 -18947.355} C_VEL
LIN {X 0,Y 249.042,Z 140.076,A -85,B 0,C 180,E1 -18952.202,E2 -18952.202} C_VEL
LIN {X 0,Y 249.045,Z 140.064,A -85,B 0,C 180,E1 -18955.64,E2 -18955.64} C_VEL
LIN {X 0,Y 249.004,Z 140.075,A -85,B 0,C 180,E1 -18959.467,E2 -18959.467} C_VEL
LIN {X 0,Y 249.027,Z 140.092,A -85,B 0,C 180,E1 -18963.157,E2 -18963.157} C_VEL
LIN {X 0,Y 249.008,Z 140.077,A -85,B 0,C 180,E1 -18966.726,E2 -18966.726} C_VEL
LIN {X 0,Y 249.103,Z 140.08,A -85,B 0,C 180,E1 -18968.949,E2 -18968.949} C_VEL
LIN {X 0,Y 249.443,Z 141.585,A -85,B 0,C 180,E1 -18969.379,E2 -18969.379} C_VEL
LIN {X 0,Y 251.664,Z 146.729,A -85,B 0,C 180,E1 -18970.993,E2 -18970.993} C_VEL
LIN {X 0,Y 260.46,Z 161.231,A -85,B 0,C 180,E1 -18973.199,E2 -18973.199} C_VEL
LIN {X 0,Y 268.582,Z 176.195,A -85,B 0,C 180,E1 -18975.132,E2 -18975.132} C_VEL
LIN {X 0,Y 275.602,Z 190.45,A -85,B 0,C 180,E1 -18976.732,E2 -18976.732} C_VEL
LIN {X 0,Y 281.136,Z 203.345,A -85,B 0,C 180,E1 -18977.969,E2 -18977.969} C_VEL
LIN {X 0,Y 275.89,Z 314.244,A -85,B 0,C 180,E1 -18980.839,E2 -18980.839} C_VEL
LIN {X 0,Y 274.467,Z 329.718,A -85,B 0,C 180,E1 -18981.487,E2 -18981.487} C_VEL
LIN {X 0,Y 272.709,Z 344.596,A -85,B 0,C 180,E1 -18982.41,E2 -18982.41} C_VEL
LIN {X 0,Y 270.701,Z 357.754,A -85,B 0,C 180,E1 -18983.478,E2 -18983.478} C_VEL
LIN {X 0,Y 268.14,Z 371.369,A -85,B 0,C 180,E1 -18984.872,E2 -18984.872} C_VEL
LIN {X 0,Y 265.258,Z 384.681,A -85,B 0,C 180,E1 -18986.582,E2 -18986.582} C_VEL
LIN {X 0,Y 262.418,Z 396.586,A -85,B 0,C 180,E1 -18988.465,E2 -18988.465} C_VEL
LIN {X 0,Y 259.321,Z 408.539,A -85,B 0,C 180,E1 -18990.782,E2 -18990.782} C_VEL
LIN {X 0,Y 256.554,Z 418.543,A -85,B 0,C 180,E1 -18993.141,E2 -18993.141} C_VEL
LIN {X 0,Y 253.867,Z 427.979,A -85,B 0,C 180,E1 -18995.85,E2 -18995.85} C_VEL
LIN {X 0,Y 251.576,Z 436.397,A -85,B 0,C 180,E1 -18998.838,E2 -18998.838} C_VEL
LIN {X 0,Y 250.044,Z 442.219,A -85,B 0,C 180,E1 -19001.347,E2 -19001.347} C_VEL
LIN {X 0,Y 248.494,Z 448.474,A -85,B 0,C 180,E1 -19004.746,E2 -19004.746} C_VEL
LIN {X 0,Y 247.448,Z 453.227,A -85,B 0,C 180,E1 -19008.205,E2 -19008.205} C_VEL
LIN {X 0,Y 246.769,Z 456.578,A -85,B 0,C 180,E1 -19011.73,E2 -19011.73} C_VEL
LIN {X 0,Y 246.474,Z 458.541,A -85,B 0,C 180,E1 -19015.322,E2 -19015.322} C_VEL
LIN {X 0,Y 246.493,Z 459.08,A -85,B 0,C 180,E1 -19017.886,E2 -19017.886} C_VEL
LIN {X 0,Y 246.705,Z 458.714,A -85,B 0,C 180,E1 -19021.28,E2 -19021.28} C_VEL
LIN {X 0,Y 247.282,Z 457.134,A -85,B 0,C 180,E1 -19024.64,E2 -19024.64} C_VEL
LIN {X 0,Y 248.091,Z 454.821,A -85,B 0,C 180,E1 -19027.514,E2 -19027.514} C_VEL
LIN {X 0,Y 249.273,Z 451.476,A -85,B 0,C 180,E1 -19030.426,E2 -19030.426} C_VEL
LIN {X 0,Y 250.806,Z 447.216,A -85,B 0,C 180,E1 -19033.233,E2 -19033.233} C_VEL
LIN {X 0,Y 252.942,Z 441.404,A -85,B 0,C 180,E1 -19036.254,E2 -19036.254} C_VEL
LIN {X 0,Y 255.77,Z 434.05,A -85,B 0,C 180,E1 -19039.27,E2 -19039.27} C_VEL
LIN {X 0,Y 258.901,Z 425.994,A -85,B 0,C 180,E1 -19041.927,E2 -19041.927} C_VEL
LIN {X 0,Y 262.015,Z 417.563,A -85,B 0,C 180,E1 -19044.232,E2 -19044.232} C_VEL
LIN {X 0,Y 265.174,Z 408.486,A -85,B 0,C 180,E1 -19046.301,E2 -19046.301} C_VEL
LIN {X 0,Y 269.106,Z 396.66,A -85,B 0,C 180,E1 -19048.511,E2 -19048.511} C_VEL
LIN {X 0,Y 272.783,Z 384.173,A -85,B 0,C 180,E1 -19050.405,E2 -19050.405} C_VEL
LIN {X 0,Y 276.174,Z 371.229,A -85,B 0,C 180,E1 -19051.98,E2 -19051.98} C_VEL
LIN {X 0,Y 277.086,Z 367.287,A -85,B 0,C 180,E1 -19052.39,E2 -19052.39} C_VEL
LIN {X 0,Y 276.87,Z 366.681,A -85,B 0,C 180,E1 -19052.515,E2 -19052.515} C_VEL
LIN {X 0,Y 263.279,Z 368.54,A -85,B 0,C 180,E1 -19054.847,E2 -19054.847} C_VEL
LIN {X 0,Y 255.529,Z 368.823,A -85,B 0,C 180,E1 -19056.496,E2 -19056.496} C_VEL
LIN {X 0,Y 254.587,Z 368.123,A -85,B 0,C 180,E1 -19056.835,E2 -19056.835} C_VEL
LIN {X 0,Y 254.168,Z 367.052,A -85,B 0,C 180,E1 -19057.117,E2 -19057.117} C_VEL
LIN {X 0,Y 252.105,Z 381.801,A -85,B 0,C 180,E1 -19059.841,E2 -19059.841} C_VEL
LIN {X 0,Y 250.911,Z 386.087,A -85,B 0,C 180,E1 -19060.728,E2 -19060.728} C_VEL
LIN {X 0,Y 247.141,Z 392.683,A -85,B 0,C 180,E1 -19062.202,E2 -19062.202} C_VEL
LIN {X 0,Y 243.447,Z 398.96,A -85,B 0,C 180,E1 -19063.793,E2 -19063.793} C_VEL
LIN {X 0,Y 242.388,Z 402.645,A -85,B 0,C 180,E1 -19064.843,E2 -19064.843} C_VEL
LIN {X 0,Y 241.28,Z 411.835,A -85,B 0,C 180,E1 -19067.808,E2 -19067.808} C_VEL
LIN {X 0,Y 240.647,Z 419.372,A -85,B 0,C 180,E1 -19070.756,E2 -19070.756} C_VEL
LIN {X 0,Y 240.282,Z 424.763,A -85,B 0,C 180,E1 -19073.281,E2 -19073.281} C_VEL
LIN {X 0,Y 240.115,Z 430.555,A -85,B 0,C 180,E1 -19076.644,E2 -19076.644} C_VEL
LIN {X 0,Y 240.095,Z 434.926,A -85,B 0,C 180,E1 -19079.999,E2 -19079.999} C_VEL
LIN {X 0,Y 240.451,Z 438.008,A -85,B 0,C 180,E1 -19083.351,E2 -19083.351} C_VEL
LIN {X 0,Y 241.031,Z 439.86,A -85,B 0,C 180,E1 -19086.697,E2 -19086.697} C_VEL
LIN {X 0,Y 242.315,Z 440.56,A -85,B 0,C 180,E1 -19090.021,E2 -19090.021} C_VEL
LIN {X 0,Y 244.136,Z 440.161,A -85,B 0,C 180,E1 -19093.314,E2 -19093.314} C_VEL
LIN {X 0,Y 246.487,Z 438.71,A -85,B 0,C 180,E1 -19096.566,E2 -19096.566} C_VEL
LIN {X 0,Y 249.797,Z 436.095,A -85,B 0,C 180,E1 -19099.731,E2 -19099.731} C_VEL
LIN {X 0,Y 253.784,Z 432.352,A -85,B 0,C 180,E1 -19102.811,E2 -19102.811} C_VEL
LIN {X 0,Y 258.591,Z 427.444,A -85,B 0,C 180,E1 -19105.775,E2 -19105.775} C_VEL
LIN {X 0,Y 264.119,Z 421.332,A -85,B 0,C 180,E1 -19108.617,E2 -19108.617} C_VEL
LIN {X 0,Y 270.352,Z 413.896,A -85,B 0,C 180,E1 -19111.326,E2 -19111.326} C_VEL
LIN {X 0,Y 277.349,Z 404.988,A -85,B 0,C 180,E1 -19113.881,E2 -19113.881} C_VEL
LIN {X 0,Y 284.971,Z 394.464,A -85,B 0,C 180,E1 -19116.291,E2 -19116.291} C_VEL
LIN {X 0,Y 292.198,Z 383.72,A -85,B 0,C 180,E1 -19118.268,E2 -19118.268} C_VEL
LIN {X 0,Y 299.98,Z 371.153,A -85,B 0,C 180,E1 -19120.111,E2 -19120.111} C_VEL
LIN {X 0,Y 307.023,Z 358.639,A -85,B 0,C 180,E1 -19121.592,E2 -19121.592} C_VEL
LIN {X 0,Y 313.838,Z 345.132,A -85,B 0,C 180,E1 -19122.86,E2 -19122.86} C_VEL
LIN {X 0,Y 320.316,Z 330.533,A -85,B 0,C 180,E1 -19123.938,E2 -19123.938} C_VEL
LIN {X 0,Y 322.776,Z 324.316,A -85,B 0,C 180,E1 -19124.321,E2 -19124.321} C_VEL
LIN {X 0,Y 323.257,Z 323.07,A -85,B 0,C 180,E1 -19124.6,E2 -19124.6} C_VEL
LIN {X 0,Y 316.439,Z 340.156,A -85,B 0,C 180,E1 -19125.45,E2 -19125.45} C_VEL
LIN {X 0,Y 308.902,Z 356.34,A -85,B 0,C 180,E1 -19126.509,E2 -19126.509} C_VEL
